KUKA KRL program: MyProgram_054().src

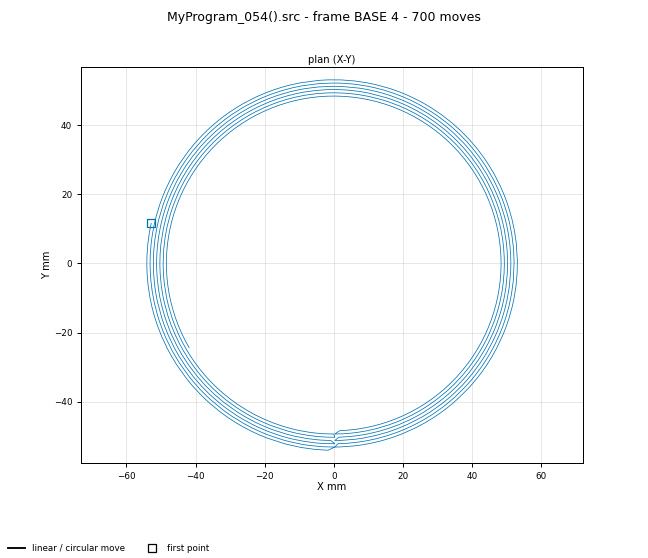
[picture p0: tool path of MyProgram_054().src in frame BASE 4, 700 of 700 moves have a stored position in this frame; points joined in program order, loops and branches not executed]
&ACCESS RVP
&REL 1
&PARAM TEMPLATE = C:\KRC\Roboter\Template\vorgabe
&PARAM EDITMASK = *
DEF MyProgram_054()
; ---- Setting reference (Base) ----
$BASE = BASE_DATA[4]

; --------------------------
; ---- Setting tool (TCP) ----
$TOOL = TOOL_DATA[3]
; --------------------------

$VEL.CP = VEL_APROX_PRINT
Startdeposition()
$VEL.CP = VEL_PRINT
LIN {X -52.8354,Y 11.6366,Z 68,A 162.012,B 24.8649,C -2.6823,E1 24.8431,E2 281.6804} C_DIS
LIN {X -53.3099,Y 9.2261,Z 68,A 164.3906,B 24.8661,C -2.6707,E1 24.8419,E2 279.3155} C_DIS
LIN {X -53.7896,Y 5.8042,Z 68,A 168.8053,B 24.8661,C -2.6709,E1 24.8404,E2 274.8737} C_DIS
LIN {X -54.0573,Y 2.193,Z 68,A 172.1652,B 24.868,C -2.6514,E1 24.8398,E2 271.5403} C_DIS
LIN {X -54.0947,Y -0.8691,Z 68,A 175.1398,B 24.8694,C -2.637,E1 24.8398,E2 268.5822} C_DIS
LIN {X -54.0113,Y -3.1274,Z 68,A 178.3127,B 24.869,C -2.6417,E1 24.8403,E2 265.379} C_DIS
LIN {X -53.6944,Y -6.6329,Z 68,A -178.5265,B 24.871,C -2.6212,E1 24.8412,E2 262.2483} C_DIS
LIN {X -53.1738,Y -9.9794,Z 68,A -174.808,B 24.8719,C -2.6123,E1 24.843,E2 258.5291} C_DIS
LIN {X -52.5931,Y -12.6871,Z 68,A -171.9255,B 24.8728,C -2.6027,E1 24.8447,E2 255.6527} C_DIS
LIN {X -51.9194,Y -15.2111,Z 68,A -168.9774,B 24.8733,C -2.5973,E1 24.847,E2 252.7003} C_DIS
LIN {X -51.0705,Y -17.8546,Z 68,A -165.794,B 24.8738,C -2.5926,E1 24.8498,E2 249.5099} C_DIS
LIN {X -49.8173,Y -21.1005,Z 68,A -162.2259,B 24.875,C -2.5803,E1 24.8536,E2 245.9513} C_DIS
LIN {X -48.2197,Y -24.5327,Z 68,A -158.7451,B 24.8769,C -2.5608,E1 24.8578,E2 242.4982} C_DIS
LIN {X -46.9289,Y -26.9196,Z 68,A -155.3829,B 24.8769,C -2.5611,E1 24.8623,E2 239.1177} C_DIS
LIN {X -45.5694,Y -29.1619,Z 68,A -152.0342,B 24.8766,C -2.5634,E1 24.8674,E2 235.7465} C_DIS
LIN {X -42.5728,Y -33.3851,Z 68,A -147.3331,B 24.8792,C -2.5373,E1 24.8751,E2 231.0852} C_DIS
LIN {X -40.8731,Y -35.4458,Z 68,A -143.9437,B 24.8789,C -2.5402,E1 24.8813,E2 227.6733} C_DIS
LIN {X -38.1407,Y -38.3706,Z 68,A -139.9381,B 24.8801,C -2.5273,E1 24.889,E2 223.6812} C_DIS
LIN {X -35.9398,Y -40.4394,Z 68,A -136.458,B 24.8802,C -2.5259,E1 24.8962,E2 220.1906} C_DIS
LIN {X -32.7163,Y -43.0888,Z 68,A -132.5105,B 24.8818,C -2.5099,E1 24.9048,E2 216.2666} C_DIS
LIN {X -30.733,Y -44.5252,Z 68,A -129.8491,B 24.882,C -2.5068,E1 24.9109,E2 213.6032} C_DIS
LIN {X -28.679,Y -45.8748,Z 68,A -127.1472,B 24.8822,C -2.5046,E1 24.9173,E2 210.8979} C_DIS
LIN {X -26.1922,Y -47.3392,Z 68,A -124.1747,B 24.8828,C -2.499,E1 24.9245,E2 207.9302} C_DIS
LIN {X -23.9334,Y -48.5199,Z 68,A -121.4558,B 24.8831,C -2.496,E1 24.9312,E2 205.2109} C_DIS
LIN {X -21.574,Y -49.614,Z 68,A -118.737,B 24.8834,C -2.4924,E1 24.9382,E2 202.4942} C_DIS
LIN {X -19.3311,Y -50.5304,Z 68,A -115.5128,B 24.8825,C -2.5019,E1 24.9466,E2 199.2404} C_DIS
LIN {X -14.037,Y -52.2489,Z 68,A -109.7546,B 24.8831,C -2.4953,E1 24.962,E2 193.4882} C_DIS
LIN {X -9.435,Y -53.2727,Z 68,A -104.9042,B 24.8836,C -2.4907,E1 24.9753,E2 188.6434} C_DIS
LIN {X -5.5823,Y -53.8128,Z 68,A -101.1152,B 24.8842,C -2.4837,E1 24.9857,E2 184.8682} C_DIS
LIN {X -1.6499,Y -54.0764,Z 68,A -96.3665,B 24.8832,C -2.495,E1 24.999,E2 180.0914} C_DIS
LIN {X -1.6499,Y -54.0764,Z 68,A -96.3665,B 24.8832,C -2.495,E1 24.999,E2 180.0914} C_DIS
Enddeposition()
LIN {X 0.3278,Y -53.1475,Z 68,A -95.9373,B 24.8845,C -2.4803,E1 25.0002,E2 179.6973} C_DIS
Startdeposition()
$VEL.CP = VEL_PRINT
LIN {X -3.2141,Y -53.0599,Z 68,A -100.1608,B 24.8853,C -2.4723,E1 24.9883,E2 183.9405} C_DIS
LIN {X -7.0942,Y -52.683,Z 68,A -104.7462,B 24.8859,C -2.466,E1 24.9755,E2 188.544} C_DIS
LIN {X -9.5086,Y -52.3006,Z 68,A -108.0099,B 24.8868,C -2.4559,E1 24.9665,E2 191.8352} C_DIS
LIN {X -12.9502,Y -51.5571,Z 68,A -110.4894,B 24.8845,C -2.4808,E1 24.9599,E2 194.2587} C_DIS
LIN {X -14.8809,Y -51.0331,Z 68,A -113.3593,B 24.8855,C -2.4697,E1 24.9521,E2 197.1596} C_DIS
LIN {X -19.1384,Y -49.5941,Z 68,A -117.5354,B 24.8841,C -2.4853,E1 24.9412,E2 201.3068} C_DIS
LIN {X -20.8488,Y -48.8986,Z 68,A -119.7452,B 24.8842,C -2.4836,E1 24.9355,E2 203.5258} C_DIS
LIN {X -23.6235,Y -47.6202,Z 68,A -122.6985,B 24.8833,C -2.4931,E1 24.9281,E2 206.4639} C_DIS
LIN {X -25.8654,Y -46.4407,Z 68,A -126.1282,B 24.8841,C -2.4849,E1 24.9196,E2 209.9228} C_DIS
LIN {X -29.6498,Y -44.1209,Z 68,A -130.8923,B 24.8834,C -2.4925,E1 24.9084,E2 214.6841} C_DIS
LIN {X -32.0346,Y -42.4208,Z 68,A -133.8914,B 24.8826,C -2.5004,E1 24.9017,E2 217.675} C_DIS
LIN {X -35.7073,Y -39.3801,Z 68,A -138.5876,B 24.8811,C -2.5172,E1 24.8917,E2 222.3493} C_DIS
LIN {X -36.9563,Y -38.2099,Z 68,A -141.2152,B 24.8819,C -2.5084,E1 24.8864,E2 225.0088} C_DIS
LIN {X -38.8214,Y -36.3135,Z 68,A -144.3826,B 24.8818,C -2.5098,E1 24.8803,E2 228.1866} C_DIS
LIN {X -41.5438,Y -33.1652,Z 68,A -149.0216,B 24.881,C -2.5177,E1 24.8721,E2 232.8282} C_DIS
LIN {X -44.6409,Y -28.8612,Z 68,A -153.9255,B 24.8785,C -2.5444,E1 24.8644,E2 237.6928} C_DIS
LIN {X -46.6361,Y -25.5121,Z 68,A -158.0676,B 24.8773,C -2.5563,E1 24.8586,E2 241.828} C_DIS
LIN {X -48.5908,Y -21.5562,Z 68,A -162.5442,B 24.8757,C -2.5736,E1 24.8532,E2 246.2874} C_DIS
LIN {X -49.5481,Y -19.255,Z 68,A -166.0559,B 24.8761,C -2.5687,E1 24.8495,E2 249.8304} C_DIS
LIN {X -50.5169,Y -16.548,Z 68,A -168.542,B 24.8744,C -2.5869,E1 24.8473,E2 252.2871} C_DIS
LIN {X -51.0383,Y -14.86,Z 68,A -170.8942,B 24.8744,C -2.5859,E1 24.8455,E2 254.6555} C_DIS
LIN {X -51.9733,Y -11.1608,Z 68,A -174.9502,B 24.8732,C -2.5991,E1 24.8429,E2 258.7036} C_DIS
LIN {X -52.5477,Y -8.0316,Z 68,A -178.1632,B 24.8718,C -2.6128,E1 24.8414,E2 261.9029} C_DIS
LIN {X -52.8915,Y -5.3189,Z 68,A 178.4615,B 24.8715,C -2.6156,E1 24.8403,E2 265.2917} C_DIS
LIN {X -53.1233,Y -1.9391,Z 68,A 175.4732,B 24.8694,C -2.6369,E1 24.8399,E2 268.2472} C_DIS
LIN {X -53.1601,Y 0.0529,Z 68,A 172.873,B 24.8694,C -2.6369,E1 24.8398,E2 270.863} C_DIS
LIN {X -53.0965,Y 2.556,Z 68,A 170.427,B 24.8682,C -2.6492,E1 24.84,E2 273.2944} C_DIS
LIN {X -52.8666,Y 5.5568,Z 68,A 166.6141,B 24.868,C -2.651,E1 24.841,E2 277.1258} C_DIS
LIN {X -52.4792,Y 8.4698,Z 68,A 163.9542,B 24.8663,C -2.6684,E1 24.8421,E2 279.7599} C_DIS
LIN {X -51.927,Y 11.3728,Z 68,A 160.5162,B 24.8657,C -2.6746,E1 24.844,E2 283.2033} C_DIS
LIN {X -51.4139,Y 13.5062,Z 68,A 157.8997,B 24.8653,C -2.6782,E1 24.8458,E2 285.8264} C_DIS
LIN {X -50.3836,Y 16.9485,Z 68,A 154.4414,B 24.8635,C -2.6962,E1 24.8487,E2 289.2616} C_DIS
LIN {X -49.6051,Y 19.1074,Z 68,A 151.9867,B 24.8627,C -2.704,E1 24.8511,E2 291.7116} C_DIS
LIN {X -48.8607,Y 20.9401,Z 68,A 149.1689,B 24.8631,C -2.7001,E1 24.8542,E2 294.5542} C_DIS
LIN {X -47.322,Y 24.2153,Z 68,A 146.0235,B 24.8608,C -2.7228,E1 24.858,E2 297.6625} C_DIS
LIN {X -45.9831,Y 26.6713,Z 68,A 142.3868,B 24.8608,C -2.722,E1 24.863,E2 301.3201} C_DIS
LIN {X -44.6959,Y 28.7757,Z 68,A 139.5821,B 24.8603,C -2.7271,E1 24.8672,E2 304.1267} C_DIS
LIN {X -41.9602,Y 32.6366,Z 68,A 134.9399,B 24.8582,C -2.7476,E1 24.8748,E2 308.7425} C_DIS
LIN {X -40.086,Y 34.9123,Z 68,A 131.5433,B 24.8577,C -2.7523,E1 24.8809,E2 312.1434} C_DIS
LIN {X -38.318,Y 36.8441,Z 68,A 129.0783,B 24.8564,C -2.7647,E1 24.8856,E2 314.5896} C_DIS
LIN {X -36.5459,Y 38.6028,Z 68,A 125.9836,B 24.8564,C -2.7647,E1 24.8918,E2 317.6972} C_DIS
LIN {X -34.6267,Y 40.3334,Z 68,A 123.5804,B 24.8552,C -2.7768,E1 24.8968,E2 320.0809} C_DIS
LIN {X -32.3135,Y 42.2093,Z 68,A 119.7034,B 24.8556,C -2.7731,E1 24.9054,E2 323.9811} C_DIS
LIN {X -30.2083,Y 43.7406,Z 68,A 117.2036,B 24.8545,C -2.7835,E1 24.9111,E2 326.4648} C_DIS
LIN {X -27.7183,Y 45.359,Z 68,A 113.9364,B 24.854,C -2.7883,E1 24.9188,E2 329.7308} C_DIS
LIN {X -25.7317,Y 46.5153,Z 68,A 111.2936,B 24.8538,C -2.7899,E1 24.9252,E2 332.3775} C_DIS
LIN {X -22.4129,Y 48.2018,Z 68,A 107.5897,B 24.8526,C -2.8011,E1 24.9345,E2 336.0642} C_DIS
LIN {X -19.7532,Y 49.3519,Z 68,A 104.3841,B 24.8523,C -2.8041,E1 24.9427,E2 339.27} C_DIS
LIN {X -17.1626,Y 50.3114,Z 68,A 101.401,B 24.8519,C -2.8077,E1 24.9506,E2 342.2505} C_DIS
LIN {X -15.0241,Y 50.9906,Z 68,A 99.3463,B 24.851,C -2.8165,E1 24.956,E2 344.2877} C_DIS
LIN {X -12.6183,Y 51.6385,Z 68,A 95.8727,B 24.8521,C -2.8058,E1 24.9655,E2 347.7918} C_DIS
LIN {X -9.8143,Y 52.2445,Z 68,A 92.5219,B 24.8523,C -2.8038,E1 24.9747,E2 351.151} C_DIS
LIN {X -4.2202,Y 52.99,Z 68,A 87.5611,B 24.8499,C -2.8266,E1 24.9883,E2 356.0607} C_DIS
LIN {X -1.6751,Y 53.1314,Z 68,A 83.82,B 24.8517,C -2.8101,E1 24.9989,E2 359.842} C_DIS
LIN {X 2.1559,Y 53.1142,Z 68,A 79.9238,B 24.8512,C -2.8147,E1 25.0097,E2 363.7266} C_DIS
LIN {X 5.9064,Y 52.8292,Z 68,A 76.491,B 24.85,C -2.8255,E1 25.0192,E2 367.1316} C_DIS
LIN {X 9.6926,Y 52.2675,Z 68,A 72.1877,B 24.8505,C -2.821,E1 25.0311,E2 371.4414} C_DIS
LIN {X 12.1047,Y 51.761,Z 68,A 69.0488,B 24.8516,C -2.8108,E1 25.0397,E2 374.6003} C_DIS
LIN {X 16.149,Y 50.646,Z 68,A 65.1105,B 24.8508,C -2.8186,E1 25.0502,E2 378.5135} C_DIS
LIN {X 17.9779,Y 50.0259,Z 68,A 63.0828,B 24.8508,C -2.8178,E1 25.0555,E2 380.5389} C_DIS
LIN {X 19.5219,Y 49.4435,Z 68,A 61.1744,B 24.8513,C -2.8137,E1 25.0605,E2 382.453} C_DIS
LIN {X 21.6172,Y 48.5645,Z 68,A 58.573,B 24.8519,C -2.8081,E1 25.0672,E2 385.0613} C_DIS
LIN {X 24.481,Y 47.1862,Z 68,A 55.3895,B 24.8519,C -2.8086,E1 25.0751,E2 388.2352} C_DIS
LIN {X 26.0526,Y 46.336,Z 68,A 53.2142,B 24.8526,C -2.8012,E1 25.0804,E2 390.4217} C_DIS
LIN {X 28.5062,Y 44.8688,Z 68,A 49.6566,B 24.8541,C -2.7873,E1 25.0889,E2 394.0008} C_DIS
LIN {X 31.3268,Y 42.9464,Z 68,A 46.1605,B 24.8543,C -2.7848,E1 25.0969,E2 397.4907} C_DIS
LIN {X 34.159,Y 40.7305,Z 68,A 42.347,B 24.8549,C -2.7789,E1 25.1051,E2 401.3037} C_DIS
LIN {X 36.7493,Y 38.4094,Z 68,A 38.7438,B 24.8554,C -2.7743,E1 25.1125,E2 404.903} C_DIS
LIN {X 39.3465,Y 35.7446,Z 68,A 34.8229,B 24.8561,C -2.7675,E1 25.12,E2 408.823} C_DIS
LIN {X 41.48,Y 33.2452,Z 68,A 31.8259,B 24.8558,C -2.7705,E1 25.1253,E2 411.7992} C_DIS
LIN {X 43.47,Y 30.5968,Z 68,A 28.2741,B 24.8567,C -2.7623,E1 25.1313,E2 415.3534} C_DIS
LIN {X 44.8639,Y 28.5132,Z 68,A 24.8197,B 24.859,C -2.74,E1 25.1366,E2 418.8433} C_DIS
LIN {X 46.3607,Y 26.0086,Z 68,A 21.4071,B 24.8604,C -2.7262,E1 25.1413,E2 422.2708} C_DIS
LIN {X 48.1892,Y 22.44,Z 68,A 18.0737,B 24.8595,C -2.7349,E1 25.1454,E2 425.5658} C_DIS
LIN {X 49.1769,Y 20.184,Z 68,A 15.2814,B 24.8606,C -2.7246,E1 25.1484,E2 428.3673} C_DIS
LIN {X 50.0014,Y 18.0457,Z 68,A 12.9638,B 24.861,C -2.7207,E1 25.1507,E2 430.6812} C_DIS
LIN {X 50.5399,Y 16.4769,Z 68,A 10.7763,B 24.8624,C -2.707,E1 25.1527,E2 432.8887} C_DIS
LIN {X 51.5927,Y 12.8059,Z 68,A 6.4948,B 24.864,C -2.6913,E1 25.1558,E2 437.1829} C_DIS
LIN {X 52.3205,Y 9.3978,Z 68,A 3.1863,B 24.8642,C -2.6893,E1 25.1576,E2 440.4767} C_DIS
LIN {X 52.8258,Y 5.9371,Z 68,A -1.0908,B 24.8664,C -2.6669,E1 25.1591,E2 444.7816} C_DIS
LIN {X 53.1526,Y 0.7627,Z 68,A -6.8833,B 24.8686,C -2.645,E1 25.1598,E2 450.5912} C_DIS
LIN {X 53.0807,Y -2.8638,Z 68,A -10.392,B 24.869,C -2.6412,E1 25.1594,E2 454.0882} C_DIS
LIN {X 52.7464,Y -6.6049,Z 68,A -14.3544,B 24.8701,C -2.6302,E1 25.1582,E2 458.053} C_DIS
LIN {X 52.1822,Y -10.1383,Z 68,A -18.1421,B 24.8712,C -2.6196,E1 25.1564,E2 461.8437} C_DIS
LIN {X 51.6671,Y -12.501,Z 68,A -20.6513,B 24.8718,C -2.6135,E1 25.1548,E2 464.3526} C_DIS
LIN {X 50.6763,Y -16.0552,Z 68,A -24.1203,B 24.8718,C -2.6121,E1 25.1521,E2 467.8053} C_DIS
LIN {X 49.8631,Y -18.425,Z 68,A -27.481,B 24.8741,C -2.5898,E1 25.1489,E2 471.1997} C_DIS
LIN {X 48.9887,Y -20.6365,Z 68,A -30.1665,B 24.8751,C -2.5796,E1 25.146,E2 473.8947} C_DIS
LIN {X 47.185,Y -24.4833,Z 68,A -34.2041,B 24.8753,C -2.5776,E1 25.1411,E2 477.9154} C_DIS
LIN {X 45.7243,Y -27.1118,Z 68,A -37.4937,B 24.8763,C -2.5674,E1 25.1365,E2 481.2121} C_DIS
LIN {X 44.4237,Y -29.1942,Z 68,A -39.8907,B 24.8765,C -2.5653,E1 25.1329,E2 483.6021} C_DIS
LIN {X 43.1358,Y -31.0663,Z 68,A -42.5014,B 24.8774,C -2.5552,E1 25.1287,E2 486.2237} C_DIS
LIN {X 41.6082,Y -33.0838,Z 68,A -45.2315,B 24.8781,C -2.548,E1 25.124,E2 488.958} C_DIS
LIN {X 40.1285,Y -34.8637,Z 68,A -47.5905,B 24.8785,C -2.5445,E1 25.1197,E2 491.3145} C_DIS
LIN {X 38.842,Y -36.2916,Z 68,A -50.2069,B 24.88,C -2.5281,E1 25.1147,E2 493.9582} C_DIS
LIN {X 35.796,Y -39.2991,Z 68,A -54.0432,B 24.8795,C -2.5333,E1 25.1071,E2 497.7664} C_DIS
LIN {X 34.3492,Y -40.5699,Z 68,A -56.2806,B 24.8803,C -2.5254,E1 25.1023,E2 500.0139} C_DIS
LIN {X 32.5435,Y -42.032,Z 68,A -58.9056,B 24.881,C -2.5175,E1 25.0966,E2 502.6475} C_DIS
LIN {X 30.4989,Y -43.5386,Z 68,A -61.6361,B 24.8815,C -2.5121,E1 25.0904,E2 505.3813} C_DIS
LIN {X 28.602,Y -44.8073,Z 68,A -63.9746,B 24.8818,C -2.5099,E1 25.0849,E2 507.7174} C_DIS
LIN {X 26.4883,Y -46.0882,Z 68,A -67.0071,B 24.8829,C -2.4977,E1 25.0775,E2 510.7694} C_DIS
LIN {X 23.8228,Y -47.5214,Z 68,A -70.3647,B 24.8836,C -2.4905,E1 25.0692,E2 514.1349} C_DIS
LIN {X 19.8322,Y -49.3203,Z 68,A -74.2061,B 24.8826,C -2.5008,E1 25.0595,E2 517.9425} C_DIS
LIN {X 16.7124,Y -50.4632,Z 68,A -78.1833,B 24.8838,C -2.4885,E1 25.049,E2 521.9409} C_DIS
LIN {X 14.0975,Y -51.2547,Z 68,A -81.1698,B 24.8841,C -2.4844,E1 25.0409,E2 524.9319} C_DIS
LIN {X 11.5851,Y -51.8807,Z 68,A -83.8242,B 24.8841,C -2.4844,E1 25.0337,E2 527.5826} C_DIS
LIN {X 8.2617,Y -52.5118,Z 68,A -87.6538,B 24.8847,C -2.478,E1 25.0232,E2 531.423} C_DIS
LIN {X 5.8899,Y -52.8303,Z 68,A -90.5802,B 24.8855,C -2.47,E1 25.015,E2 534.3663} C_DIS
LIN {X 1.7317,Y -53.1297,Z 68,A -94.4063,B 24.8845,C -2.4805,E1 25.0044,E2 538.1659} C_DIS
LIN {X 0.3278,Y -53.1475,Z 68,A -95.9366,B 24.8845,C -2.48,E1 25.0002,E2 539.6973} C_DIS
Enddeposition()
LIN {X 0.3278,Y -53.1475,Z 68,A -95.9366,B 24.8845,C -2.48,E1 25.0002,E2 539.6973} C_DIS
Startdeposition()
$VEL.CP = VEL_PRINT
LIN {X 1.2007,Y -52.2008,Z 68,A -93.7724,B 24.8809,C -2.5188,E1 25.0065,E2 537.4412} C_DIS
LIN {X 3.7036,Y -52.0819,Z 68,A -91.0856,B 24.8809,C -2.5188,E1 25.0139,E2 534.7556} C_DIS
LIN {X 6.9902,Y -51.7448,Z 68,A -87.899,B 24.8815,C -2.5126,E1 25.0227,E2 531.5859} C_DIS
LIN {X 9.5939,Y -51.3254,Z 68,A -84.4131,B 24.8802,C -2.5261,E1 25.0324,E2 528.0716} C_DIS
LIN {X 12.2252,Y -50.763,Z 68,A -81.8964,B 24.8808,C -2.5204,E1 25.0392,E2 525.5718} C_DIS
LIN {X 15.4906,Y -49.8633,Z 68,A -78.0208,B 24.8801,C -2.5276,E1 25.0496,E2 521.6859} C_DIS
LIN {X 18.3377,Y -48.8883,Z 68,A -74.7631,B 24.8798,C -2.5309,E1 25.0582,E2 518.4269} C_DIS
LIN {X 20.4504,Y -48.0429,Z 68,A -72.3518,B 24.8796,C -2.5327,E1 25.0644,E2 516.0168} C_DIS
LIN {X 22.4531,Y -47.1401,Z 68,A -69.8259,B 24.879,C -2.5387,E1 25.0708,E2 513.4832} C_DIS
LIN {X 24.1625,Y -46.2874,Z 68,A -67.9284,B 24.879,C -2.5382,E1 25.0755,E2 511.5921} C_DIS
LIN {X 26.2875,Y -45.1148,Z 68,A -65.0106,B 24.8781,C -2.548,E1 25.0826,E2 508.6599} C_DIS
LIN {X 28.7287,Y -43.6001,Z 68,A -61.8105,B 24.8775,C -2.5549,E1 25.0902,E2 505.4537} C_DIS
LIN {X 31.3281,Y -41.7715,Z 68,A -58.6989,B 24.8775,C -2.5543,E1 25.0972,E2 502.3545} C_DIS
LIN {X 32.8885,Y -40.5544,Z 68,A -55.8361,B 24.8757,C -2.5732,E1 25.1035,E2 499.4578} C_DIS
LIN {X 35.0118,Y -38.7368,Z 68,A -52.7354,B 24.875,C -2.5808,E1 25.11,E2 496.3514} C_DIS
LIN {X 38.2717,Y -35.5199,Z 68,A -48.6469,B 24.8757,C -2.5734,E1 25.1179,E2 492.2979} C_DIS
LIN {X 40.1139,Y -33.4244,Z 68,A -45.4119,B 24.8746,C -2.5848,E1 25.1238,E2 489.0506} C_DIS
LIN {X 41.3473,Y -31.8858,Z 68,A -42.9646,B 24.8734,C -2.5964,E1 25.1281,E2 486.5874} C_DIS
LIN {X 43.203,Y -29.3225,Z 68,A -39.5516,B 24.8726,C -2.6045,E1 25.1336,E2 483.1718} C_DIS
LIN {X 44.7418,Y -26.9172,Z 68,A -36.3924,B 24.8717,C -2.6138,E1 25.1382,E2 480.0067} C_DIS
LIN {X 45.9347,Y -24.8258,Z 68,A -34.2432,B 24.872,C -2.611,E1 25.1411,E2 477.8754} C_DIS
LIN {X 46.8178,Y -23.1172,Z 68,A -31.8383,B 24.8708,C -2.6233,E1 25.1442,E2 475.454} C_DIS
LIN {X 48.0762,Y -20.3714,Z 68,A -28.7816,B 24.8704,C -2.6277,E1 25.1476,E2 472.4037} C_DIS
LIN {X 48.9685,Y -18.1232,Z 68,A -25.588,B 24.8684,C -2.6472,E1 25.1508,E2 469.1817} C_DIS
LIN {X 49.8838,Y -15.4247,Z 68,A -22.5315,B 24.8676,C -2.6553,E1 25.1534,E2 466.1234} C_DIS
LIN {X 50.6755,Y -12.5838,Z 68,A -19.3049,B 24.8666,C -2.6651,E1 25.1557,E2 462.8921} C_DIS
LIN {X 51.4366,Y -8.9803,Z 68,A -15.5277,B 24.8659,C -2.6721,E1 25.1577,E2 459.1205} C_DIS
LIN {X 51.9731,Y -5.0149,Z 68,A -10.3276,B 24.8628,C -2.7034,E1 25.1594,E2 453.8772} C_DIS
LIN {X 52.2139,Y 0.3513,Z 68,A -4.5685,B 24.8612,C -2.719,E1 25.1597,E2 448.1154} C_DIS
LIN {X 52.0275,Y 4.4168,Z 68,A -0.3147,B 24.8602,C -2.7283,E1 25.1589,E2 443.8647} C_DIS
LIN {X 51.5536,Y 8.2844,Z 68,A 3.549,B 24.8597,C -2.7327,E1 25.1573,E2 440.0135} C_DIS
LIN {X 50.8864,Y 11.6998,Z 68,A 7.0648,B 24.8592,C -2.7379,E1 25.1553,E2 436.5059} C_DIS
LIN {X 50.2849,Y 14.0622,Z 68,A 10.0343,B 24.8577,C -2.7521,E1 25.1532,E2 433.5198} C_DIS
LIN {X 49.4397,Y 16.7941,Z 68,A 12.8575,B 24.8575,C -2.7546,E1 25.1507,E2 430.7066} C_DIS
LIN {X 48.7669,Y 18.6582,Z 68,A 14.8622,B 24.8572,C -2.7573,E1 25.1488,E2 428.7068} C_DIS
LIN {X 47.7195,Y 21.1952,Z 68,A 18.4495,B 24.8551,C -2.7779,E1 25.1448,E2 425.0905} C_DIS
LIN {X 46.144,Y 24.4343,Z 68,A 22.4166,B 24.8539,C -2.7889,E1 25.1398,E2 421.1184} C_DIS
LIN {X 44.0565,Y 28.0234,Z 68,A 26.713,B 24.8532,C -2.7952,E1 25.1336,E2 416.8288} C_DIS
LIN {X 42.4536,Y 30.3974,Z 68,A 30.2406,B 24.8516,C -2.8109,E1 25.1279,E2 413.2813} C_DIS
LIN {X 40.5493,Y 32.8947,Z 68,A 33.4134,B 24.8513,C -2.8133,E1 25.1224,E2 410.1177} C_DIS
LIN {X 38.6742,Y 35.0814,Z 68,A 36.2791,B 24.8513,C -2.8143,E1 25.1171,E2 407.2625} C_DIS
LIN {X 36.2281,Y 37.601,Z 68,A 39.8075,B 24.8511,C -2.8158,E1 25.1102,E2 403.7455} C_DIS
LIN {X 34.4102,Y 39.2715,Z 68,A 42.7374,B 24.85,C -2.8255,E1 25.1041,E2 400.8043} C_DIS
LIN {X 32.7671,Y 40.6527,Z 68,A 45.8391,B 24.848,C -2.8448,E1 25.0973,E2 397.6687} C_DIS
LIN {X 29.8757,Y 42.8224,Z 68,A 49.1443,B 24.8487,C -2.8383,E1 25.0898,E2 394.3905} C_DIS
LIN {X 27.988,Y 44.08,Z 68,A 51.7817,B 24.8479,C -2.845,E1 25.0836,E2 391.7458} C_DIS
LIN {X 24.7155,Y 45.9945,Z 68,A 55.7511,B 24.8477,C -2.847,E1 25.074,E2 387.7834} C_DIS
LIN {X 22.1577,Y 47.2796,Z 68,A 58.8989,B 24.8473,C -2.8509,E1 25.0661,E2 384.6346} C_DIS
LIN {X 19.7851,Y 48.3205,Z 68,A 61.7258,B 24.847,C -2.8535,E1 25.0588,E2 381.8082} C_DIS
LIN {X 17.2309,Y 49.289,Z 68,A 64.6932,B 24.8468,C -2.8557,E1 25.051,E2 378.842} C_DIS
LIN {X 14.4825,Y 50.1661,Z 68,A 67.922,B 24.8464,C -2.8591,E1 25.0424,E2 375.6106} C_DIS
LIN {X 11.9937,Y 50.8176,Z 68,A 70.7137,B 24.8464,C -2.8602,E1 25.0348,E2 372.8206} C_DIS
LIN {X 10.021,Y 51.2436,Z 68,A 72.93,B 24.8462,C -2.8611,E1 25.0288,E2 370.6046} C_DIS
LIN {X 6.9548,Y 51.7494,Z 68,A 76.043,B 24.8467,C -2.8567,E1 25.0202,E2 367.5052} C_DIS
LIN {X 5.4409,Y 51.9298,Z 68,A 78.0087,B 24.8461,C -2.8622,E1 25.0147,E2 365.5277} C_DIS
LIN {X 2.4355,Y 52.1576,Z 68,A 81.2381,B 24.8462,C -2.8608,E1 25.0057,E2 362.3029} C_DIS
LIN {X -0.237,Y 52.2136,Z 68,A 84.7379,B 24.8452,C -2.8704,E1 24.9959,E2 358.7805} C_DIS
LIN {X -4.4458,Y 52.0252,Z 68,A 89.4616,B 24.8452,C -2.8703,E1 24.9827,E2 354.0553} C_DIS
LIN {X -9.1801,Y 51.4008,Z 68,A 94.127,B 24.8467,C -2.8568,E1 24.9699,E2 349.4181} C_DIS
LIN {X -11.9273,Y 50.8339,Z 68,A 97.6428,B 24.8461,C -2.8616,E1 24.9603,E2 345.8863} C_DIS
LIN {X -14.9887,Y 50.0164,Z 68,A 100.8953,B 24.847,C -2.8541,E1 24.9516,E2 342.6464} C_DIS
LIN {X -18.2145,Y 48.9347,Z 68,A 104.3166,B 24.848,C -2.8443,E1 24.9427,E2 339.2418} C_DIS
LIN {X -20.4534,Y 48.0417,Z 68,A 106.8717,B 24.8486,C -2.8392,E1 24.9361,E2 336.6932} C_DIS
LIN {X -22.2243,Y 47.2486,Z 68,A 109.6359,B 24.8478,C -2.8464,E1 24.929,E2 333.9047} C_DIS
LIN {X -25.0712,Y 45.8016,Z 68,A 112.3861,B 24.8497,C -2.8284,E1 24.9223,E2 331.19} C_DIS
LIN {X -26.937,Y 44.7298,Z 68,A 116.0793,B 24.8478,C -2.8458,E1 24.9133,E2 327.4439} C_DIS
LIN {X -29.6438,Y 42.9836,Z 68,A 118.1309,B 24.8511,C -2.8152,E1 24.9087,E2 325.4587} C_DIS
LIN {X -31.4396,Y 41.6877,Z 68,A 121.0877,B 24.8508,C -2.8186,E1 24.902,E2 322.4831} C_DIS
LIN {X -33.7792,Y 39.8156,Z 68,A 123.8326,B 24.8524,C -2.803,E1 24.8962,E2 319.7651} C_DIS
LIN {X -35.8205,Y 37.9895,Z 68,A 127.8827,B 24.8514,C -2.8126,E1 24.8877,E2 315.6758} C_DIS
LIN {X -37.868,Y 35.9497,Z 68,A 131.1106,B 24.8521,C -2.8058,E1 24.8815,E2 312.4501} C_DIS
LIN {X -40.9903,Y 32.3435,Z 68,A 135.348,B 24.8551,C -2.7772,E1 24.874,E2 308.2618} C_DIS
LIN {X -42.5301,Y 30.2902,Z 68,A 139.0655,B 24.8545,C -2.7835,E1 24.8678,E2 304.5112} C_DIS
LIN {X -44.1197,Y 27.9252,Z 68,A 142.0352,B 24.8556,C -2.7725,E1 24.8633,E2 301.5529} C_DIS
LIN {X -45.9239,Y 24.8457,Z 68,A 145.4828,B 24.8575,C -2.7543,E1 24.8586,E2 298.1307} C_DIS
LIN {X -46.9052,Y 22.941,Z 68,A 148.4228,B 24.8573,C -2.7563,E1 24.8549,E2 295.17} C_DIS
LIN {X -47.9109,Y 20.7573,Z 68,A 150.8147,B 24.8585,C -2.7448,E1 24.8522,E2 292.7925} C_DIS
LIN {X -48.8857,Y 18.3442,Z 68,A 153.3925,B 24.8598,C -2.7321,E1 24.8496,E2 290.2306} C_DIS
LIN {X -49.4483,Y 16.7684,Z 68,A 155.9091,B 24.8593,C -2.7367,E1 24.8473,E2 287.6888} C_DIS
LIN {X -50.6514,Y 12.6825,Z 68,A 160.5516,B 24.8609,C -2.7218,E1 24.8439,E2 283.0549} C_DIS
LIN {X -51.3189,Y 9.6282,Z 68,A 163.7038,B 24.8624,C -2.7069,E1 24.8422,E2 279.9197} C_DIS
LIN {X -51.7597,Y 6.872,Z 68,A 166.8961,B 24.8632,C -2.6992,E1 24.8409,E2 276.7267} C_DIS
LIN {X -52.0814,Y 3.7254,Z 68,A 170.2384,B 24.8645,C -2.6864,E1 24.8401,E2 273.3951} C_DIS
LIN {X -52.2046,Y 0.9956,Z 68,A 173.6641,B 24.8648,C -2.6833,E1 24.8398,E2 269.9562} C_DIS
LIN {X -52.1647,Y -2.2699,Z 68,A 176.8993,B 24.8664,C -2.6668,E1 24.84,E2 266.7408} C_DIS
LIN {X -51.8799,Y -5.9007,Z 68,A -178.518,B 24.8668,C -2.6632,E1 24.8413,E2 262.1393} C_DIS
LIN {X -51.4684,Y -8.7948,Z 68,A -175.7448,B 24.8685,C -2.6468,E1 24.8425,E2 259.3888} C_DIS
LIN {X -51.0492,Y -10.969,Z 68,A -172.8105,B 24.8685,C -2.6471,E1 24.8442,E2 256.4367} C_DIS
LIN {X -49.7332,Y -15.9045,Z 68,A -168.2663,B 24.8717,C -2.6144,E1 24.8476,E2 251.9443} C_DIS
LIN {X -49.045,Y -17.9137,Z 68,A -164.7943,B 24.8706,C -2.625,E1 24.8509,E2 248.4273} C_DIS
LIN {X -47.8972,Y -20.7889,Z 68,A -161.0104,B 24.871,C -2.6214,E1 24.8551,E2 244.6309} C_DIS
LIN {X -46.075,Y -24.5656,Z 68,A -157.3797,B 24.8737,C -2.5939,E1 24.8597,E2 241.0467} C_DIS
LIN {X -44.7087,Y -26.9716,Z 68,A -154.0153,B 24.874,C -2.5911,E1 24.8644,E2 237.6714} C_DIS
LIN {X -42.7042,Y -30.0458,Z 68,A -149.0279,B 24.8734,C -2.5964,E1 24.8724,E2 232.6467} C_DIS
LIN {X -40.5227,Y -32.9275,Z 68,A -145.9912,B 24.8758,C -2.5723,E1 24.8776,E2 229.6534} C_DIS
LIN {X -38.1501,Y -35.6498,Z 68,A -142.8037,B 24.8778,C -2.5512,E1 24.8835,E2 226.5019} C_DIS
LIN {X -35.759,Y -38.0474,Z 68,A -139.1122,B 24.8786,C -2.5432,E1 24.8908,E2 222.814} C_DIS
LIN {X -32.9352,Y -40.5165,Z 68,A -134.8843,B 24.8792,C -2.5371,E1 24.8997,E2 218.584} C_DIS
LIN {X -30.8948,Y -42.093,Z 68,A -131.4388,B 24.8787,C -2.5424,E1 24.9074,E2 215.1136} C_DIS
LIN {X -27.9737,Y -44.0892,Z 68,A -128.0415,B 24.88,C -2.5282,E1 24.9153,E2 211.7388} C_DIS
LIN {X -26.3271,Y -45.0918,Z 68,A -125.4385,B 24.8795,C -2.5334,E1 24.9216,E2 209.1155} C_DIS
LIN {X -23.6104,Y -46.5713,Z 68,A -122.6543,B 24.8809,C -2.5188,E1 24.9284,E2 206.3585} C_DIS
LIN {X -21.6547,Y -47.5124,Z 68,A -119.5684,B 24.88,C -2.5281,E1 24.9362,E2 203.2426} C_DIS
LIN {X -18.9453,Y -48.656,Z 68,A -116.3556,B 24.8803,C -2.5247,E1 24.9446,E2 200.0307} C_DIS
LIN {X -15.9666,Y -49.7127,Z 68,A -113.1831,B 24.8811,C -2.5168,E1 24.9529,E2 196.8711} C_DIS
LIN {X -13.608,Y -50.4096,Z 68,A -110.7445,B 24.8817,C -2.5105,E1 24.9594,E2 194.4436} C_DIS
LIN {X -11.8411,Y -50.8538,Z 68,A -107.9542,B 24.8805,C -2.5235,E1 24.9671,E2 191.6185} C_DIS
LIN {X -8.6106,Y -51.4992,Z 68,A -104.6005,B 24.881,C -2.5176,E1 24.9763,E2 188.2754} C_DIS
LIN {X -5.2253,Y -51.9524,Z 68,A -101.3512,B 24.8819,C -2.5079,E1 24.9852,E2 185.0468} C_DIS
LIN {X -3.3589,Y -52.1062,Z 68,A -98.5237,B 24.8806,C -2.5221,E1 24.9932,E2 182.1846} C_DIS
LIN {X 0.3319,Y -52.2067,Z 68,A -96.1542,B 24.8834,C -2.492,E1 24.9996,E2 179.8863} C_DIS
Enddeposition()
LIN {X 0.3319,Y -52.2067,Z 68,A -96.1542,B 24.8834,C -2.492,E1 24.9996,E2 179.8863} C_DIS
Startdeposition()
$VEL.CP = VEL_PRINT
LIN {X -0.8087,Y -51.2641,Z 68,A -97.7461,B 24.8824,C -2.5026,E1 24.9952,E2 181.4532} C_DIS
LIN {X -3.7459,Y -51.1341,Z 68,A -100.8536,B 24.8822,C -2.5056,E1 24.9866,E2 184.5545} C_DIS
LIN {X -5.5282,Y -50.9717,Z 68,A -102.9078,B 24.8822,C -2.5048,E1 24.9809,E2 186.6117} C_DIS
LIN {X -8.0735,Y -50.6311,Z 68,A -106.1583,B 24.8828,C -2.499,E1 24.9719,E2 189.8789} C_DIS
LIN {X -11.4791,Y -49.9688,Z 68,A -109.6591,B 24.882,C -2.5071,E1 24.9623,E2 193.3647} C_DIS
LIN {X -13.4357,Y -49.4786,Z 68,A -112.2716,B 24.8825,C -2.5024,E1 24.9553,E2 195.9923} C_DIS
LIN {X -17.0996,Y -48.3348,Z 68,A -115.8765,B 24.8811,C -2.5171,E1 24.9458,E2 199.5688} C_DIS
LIN {X -18.7522,Y -47.7179,Z 68,A -117.8059,B 24.8808,C -2.5196,E1 24.9407,E2 201.4964} C_DIS
LIN {X -20.8732,Y -46.8294,Z 68,A -120.9009,B 24.8814,C -2.5136,E1 24.9327,E2 204.6128} C_DIS
LIN {X -23.1559,Y -45.7437,Z 68,A -123.7032,B 24.881,C -2.5173,E1 24.9257,E2 207.4135} C_DIS
LIN {X -25.6921,Y -44.3688,Z 68,A -126.8217,B 24.8805,C -2.5234,E1 24.9182,E2 210.5268} C_DIS
LIN {X -28.124,Y -42.8684,Z 68,A -130.8298,B 24.8812,C -2.5154,E1 24.9087,E2 214.5668} C_DIS
LIN {X -31.806,Y -40.2123,Z 68,A -134.6994,B 24.8786,C -2.5428,E1 24.9001,E2 218.3848} C_DIS
LIN {X -34.5688,Y -37.8636,Z 68,A -138.9491,B 24.8782,C -2.5474,E1 24.8911,E2 222.6402} C_DIS
LIN {X -37.0936,Y -35.3946,Z 68,A -142.748,B 24.8772,C -2.5578,E1 24.8836,E2 226.4303} C_DIS
LIN {X -39.3761,Y -32.8356,Z 68,A -146.9834,B 24.877,C -2.5602,E1 24.8758,E2 230.6791} C_DIS
LIN {X -42.0224,Y -29.3732,Z 68,A -151.8997,B 24.8759,C -2.5711,E1 24.8676,E2 235.5929} C_DIS
LIN {X -43.9944,Y -26.3289,Z 68,A -156.0437,B 24.875,C -2.5801,E1 24.8615,E2 239.7365} C_DIS
LIN {X -45.32,Y -23.9739,Z 68,A -158.8961,B 24.874,C -2.5906,E1 24.8577,E2 242.5789} C_DIS
LIN {X -46.8687,Y -20.7849,Z 68,A -162.6411,B 24.8726,C -2.6047,E1 24.8532,E2 246.3106} C_DIS
LIN {X -47.4227,Y -19.4873,Z 68,A -165.3906,B 24.8738,C -2.5922,E1 24.8502,E2 249.1052} C_DIS
LIN {X -48.7728,Y -15.8068,Z 68,A -168.8073,B 24.8712,C -2.6187,E1 24.8472,E2 252.478} C_DIS
LIN {X -49.6569,Y -12.7608,Z 68,A -172.9324,B 24.871,C -2.621,E1 24.8441,E2 256.6216} C_DIS
LIN {X -50.3229,Y -9.808,Z 68,A -176.1319,B 24.8697,C -2.6339,E1 24.8423,E2 259.8092} C_DIS
LIN {X -50.7273,Y -7.4458,Z 68,A -179.8186,B 24.8703,C -2.628,E1 24.8408,E2 263.5319} C_DIS
LIN {X -51.1133,Y -4.0099,Z 68,A 177.5359,B 24.8674,C -2.657,E1 24.8401,E2 266.1238} C_DIS
LIN {X -51.2514,Y -1.4029,Z 68,A 174.6766,B 24.8664,C -2.667,E1 24.8398,E2 268.9765} C_DIS
LIN {X -51.2622,Y 0.9094,Z 68,A 172.0803,B 24.8656,C -2.675,E1 24.8398,E2 271.5694} C_DIS
LIN {X -51.1841,Y 2.9757,Z 68,A 169.7958,B 24.8649,C -2.6826,E1 24.8401,E2 273.8494} C_DIS
LIN {X -51.0191,Y 5.0758,Z 68,A 167.326,B 24.8643,C -2.6884,E1 24.8407,E2 276.3202} C_DIS
LIN {X -50.644,Y 7.9911,Z 68,A 163.6039,B 24.8639,C -2.6926,E1 24.8422,E2 280.0545} C_DIS
LIN {X -50.1036,Y 10.8755,Z 68,A 160.7027,B 24.8623,C -2.7081,E1 24.8438,E2 282.9356} C_DIS
LIN {X -49.602,Y 12.9745,Z 68,A 158.3301,B 24.8614,C -2.7161,E1 24.8454,E2 285.303} C_DIS
LIN {X -48.9598,Y 15.218,Z 68,A 155.4965,B 24.861,C -2.721,E1 24.8477,E2 288.1413} C_DIS
LIN {X -48.163,Y 17.5775,Z 68,A 152.3392,B 24.8606,C -2.7241,E1 24.8507,E2 291.3089} C_DIS
LIN {X -47.0789,Y 20.3041,Z 68,A 149.1581,B 24.8595,C -2.7352,E1 24.8541,E2 294.4811} C_DIS
LIN {X -45.7787,Y 23.0874,Z 68,A 145.9999,B 24.858,C -2.7491,E1 24.8579,E2 297.6231} C_DIS
LIN {X -44.9116,Y 24.732,Z 68,A 143.8214,B 24.8576,C -2.7536,E1 24.8608,E2 299.8024} C_DIS
LIN {X -43.5554,Y 27.048,Z 68,A 141.1218,B 24.8563,C -2.7663,E1 24.8647,E2 302.4855} C_DIS
LIN {X -42.6401,Y 28.4702,Z 68,A 139.0175,B 24.856,C -2.7684,E1 24.8679,E2 304.5954} C_DIS
LIN {X -40.9737,Y 30.8188,Z 68,A 135.7117,B 24.8553,C -2.7757,E1 24.8733,E2 307.8999} C_DIS
LIN {X -38.5495,Y 33.8022,Z 68,A 131.0811,B 24.8547,C -2.7817,E1 24.8817,E2 312.5374} C_DIS
LIN {X -36.7313,Y 35.7705,Z 68,A 128.1852,B 24.8537,C -2.7904,E1 24.8872,E2 315.4252} C_DIS
LIN {X -33.9447,Y 38.4251,Z 68,A 124.0239,B 24.8525,C -2.8022,E1 24.8957,E2 319.575} C_DIS
LIN {X -31.1612,Y 40.7136,Z 68,A 119.7751,B 24.8519,C -2.8074,E1 24.905,E2 323.8272} C_DIS
LIN {X -29.0309,Y 42.2596,Z 68,A 117.229,B 24.8507,C -2.8192,E1 24.9108,E2 326.3539} C_DIS
LIN {X -27.0508,Y 43.5536,Z 68,A 114.453,B 24.8504,C -2.8221,E1 24.9173,E2 329.1319} C_DIS
LIN {X -24.7912,Y 44.8787,Z 68,A 111.7908,B 24.8494,C -2.8313,E1 24.9237,E2 331.7802} C_DIS
LIN {X -22.5297,Y 46.0557,Z 68,A 108.9982,B 24.8488,C -2.8367,E1 24.9307,E2 334.5673} C_DIS
LIN {X -20.7937,Y 46.8647,Z 68,A 106.5471,B 24.849,C -2.835,E1 24.9369,E2 337.0285} C_DIS
LIN {X -18.8412,Y 47.6829,Z 68,A 104.345,B 24.8484,C -2.8408,E1 24.9426,E2 339.2216} C_DIS
LIN {X -16.2126,Y 48.6398,Z 68,A 100.5211,B 24.8492,C -2.8335,E1 24.9527,E2 343.0704} C_DIS
LIN {X -12.7282,Y 49.6653,Z 68,A 96.9641,B 24.8479,C -2.8458,E1 24.9623,E2 346.6038} C_DIS
LIN {X -10.3193,Y 50.2211,Z 68,A 94.1397,B 24.8477,C -2.8471,E1 24.97,E2 349.4284} C_DIS
LIN {X -8.2819,Y 50.5973,Z 68,A 91.5954,B 24.8479,C -2.845,E1 24.977,E2 351.9802} C_DIS
LIN {X -4.4591,Y 51.0767,Z 68,A 86.5266,B 24.849,C -2.8346,E1 24.9911,E2 357.0765} C_DIS
LIN {X -0.0283,Y 51.271,Z 68,A 82.5726,B 24.8471,C -2.8528,E1 25.0021,E2 360.9877} C_DIS
LIN {X 2.4813,Y 51.211,Z 68,A 79.0899,B 24.8483,C -2.8414,E1 25.0118,E2 364.4966} C_DIS
LIN {X 7.4712,Y 50.7237,Z 68,A 74.156,B 24.8472,C -2.852,E1 25.0254,E2 369.4015} C_DIS
LIN {X 9.9052,Y 50.3048,Z 68,A 71.754,B 24.8466,C -2.8573,E1 25.032,E2 371.7883} C_DIS
LIN {X 12.4115,Y 49.7454,Z 68,A 68.2518,B 24.848,C -2.8446,E1 25.0416,E2 375.3158} C_DIS
LIN {X 14.8769,Y 49.0647,Z 68,A 65.8404,B 24.8473,C -2.8506,E1 25.048,E2 377.7088} C_DIS
LIN {X 16.4811,Y 48.5492,Z 68,A 63.5097,B 24.8484,C -2.841,E1 25.0542,E2 380.0579} C_DIS
LIN {X 20.1701,Y 47.1369,Z 68,A 59.7601,B 24.8475,C -2.8488,E1 25.0639,E2 383.7805} C_DIS
LIN {X 22.4437,Y 46.0977,Z 68,A 56.5745,B 24.8486,C -2.8384,E1 25.072,E2 386.9828} C_DIS
LIN {X 24.744,Y 44.905,Z 68,A 53.3742,B 24.8497,C -2.8289,E1 25.0799,E2 390.1964} C_DIS
LIN {X 27.4699,Y 43.2911,Z 68,A 49.8931,B 24.8501,C -2.8247,E1 25.0882,E2 393.6764} C_DIS
LIN {X 29.9782,Y 41.5934,Z 68,A 46.6007,B 24.8505,C -2.8209,E1 25.0957,E2 396.9665} C_DIS
LIN {X 32.5407,Y 39.6212,Z 68,A 43.4095,B 24.8503,C -2.8225,E1 25.1026,E2 400.142} C_DIS
LIN {X 34.7073,Y 37.7366,Z 68,A 40.0572,B 24.8513,C -2.8135,E1 25.1097,E2 403.5022} C_DIS
LIN {X 37.6447,Y 34.8074,Z 68,A 35.5629,B 24.852,C -2.8066,E1 25.1185,E2 407.9939} C_DIS
LIN {X 39.7733,Y 32.3534,Z 68,A 31.9889,B 24.8528,C -2.7994,E1 25.1249,E2 411.5684} C_DIS
LIN {X 41.434,Y 30.1974,Z 68,A 28.9725,B 24.8535,C -2.7927,E1 25.13,E2 414.5865} C_DIS
LIN {X 42.4862,Y 28.698,Z 68,A 26.2861,B 24.8554,C -2.7749,E1 25.1343,E2 417.3017} C_DIS
LIN {X 44.3654,Y 25.698,Z 68,A 22.2803,B 24.8565,C -2.7637,E1 25.14,E2 421.3137} C_DIS
LIN {X 46.1778,Y 22.277,Z 68,A 18.7732,B 24.856,C -2.7684,E1 25.1445,E2 424.791} C_DIS
LIN {X 47.2402,Y 19.9252,Z 68,A 15.6277,B 24.8574,C -2.755,E1 25.148,E2 427.9509} C_DIS
LIN {X 48.129,Y 17.6706,Z 68,A 12.1343,B 24.8599,C -2.7314,E1 25.1514,E2 431.4807} C_DIS
LIN {X 49.4435,Y 13.5654,Z 68,A 8.127,B 24.8597,C -2.7336,E1 25.1546,E2 435.46} C_DIS
LIN {X 50.0822,Y 10.9737,Z 68,A 5.0214,B 24.8608,C -2.7221,E1 25.1566,E2 438.5748} C_DIS
LIN {X 50.5941,Y 8.3011,Z 68,A 2.1699,B 24.8614,C -2.7166,E1 25.158,E2 441.4225} C_DIS
LIN {X 50.9961,Y 5.2956,Z 68,A -1.2446,B 24.8625,C -2.7056,E1 25.1591,E2 444.8429} C_DIS
LIN {X 51.2094,Y 2.517,Z 68,A -3.9853,B 24.8627,C -2.7035,E1 25.1596,E2 447.5722} C_DIS
LIN {X 51.273,Y -0.0468,Z 68,A -7.5888,B 24.8652,C -2.6793,E1 25.1597,E2 451.2115} C_DIS
LIN {X 51.218,Y -2.3185,Z 68,A -10.2622,B 24.8663,C -2.6686,E1 25.1594,E2 453.8944} C_DIS
LIN {X 50.7461,Y -7.3139,Z 68,A -15.2768,B 24.8668,C -2.6631,E1 25.1578,E2 458.8924} C_DIS
LIN {X 50.078,Y -10.9918,Z 68,A -19.6072,B 24.8684,C -2.6469,E1 25.1555,E2 463.2358} C_DIS
LIN {X 49.4645,Y -13.4877,Z 68,A -22.3393,B 24.869,C -2.6408,E1 25.1536,E2 465.9665} C_DIS
LIN {X 48.6396,Y -16.213,Z 68,A -26.1315,B 24.8713,C -2.6186,E1 25.1503,E2 469.7897} C_DIS
LIN {X 47.4277,Y -19.4751,Z 68,A -28.9406,B 24.8702,C -2.629,E1 25.1475,E2 472.5587} C_DIS
LIN {X 46.3211,Y -21.9762,Z 68,A -32.8582,B 24.8728,C -2.6024,E1 25.1429,E2 476.518} C_DIS
LIN {X 44.1395,Y -26.0835,Z 68,A -37.9181,B 24.874,C -2.5903,E1 25.136,E2 481.5801} C_DIS
LIN {X 42.5304,Y -28.6327,Z 68,A -41.1614,B 24.8747,C -2.5836,E1 25.131,E2 484.8231} C_DIS
LIN {X 40.2989,Y -31.6963,Z 68,A -45.0626,B 24.8751,C -2.5791,E1 25.1244,E2 488.7164} C_DIS
LIN {X 38.4358,Y -33.9318,Z 68,A -48.1128,B 24.8755,C -2.5749,E1 25.1189,E2 491.7627} C_DIS
LIN {X 37.1523,Y -35.3324,Z 68,A -50.5888,B 24.8767,C -2.5626,E1 25.1141,E2 494.2569} C_DIS
LIN {X 34.8216,Y -37.6317,Z 68,A -53.8272,B 24.8767,C -2.5624,E1 25.1076,E2 497.4823} C_DIS
LIN {X 33.4009,Y -38.8978,Z 68,A -56.2661,B 24.8778,C -2.5515,E1 25.1025,E2 499.9376} C_DIS
LIN {X 31.1355,Y -40.734,Z 68,A -59.6725,B 24.8787,C -2.5417,E1 25.095,E2 503.3546} C_DIS
LIN {X 28.0259,Y -42.9331,Z 68,A -63.3691,B 24.8785,C -2.5442,E1 25.0865,E2 507.0326} C_DIS
LIN {X 25.4695,Y -44.4967,Z 68,A -67.5016,B 24.8805,C -2.5231,E1 25.0765,E2 511.2025} C_DIS
LIN {X 21.125,Y -46.716,Z 68,A -72.8313,B 24.8811,C -2.5168,E1 25.0631,E2 516.5329} C_DIS
LIN {X 18.2951,Y -47.8947,Z 68,A -75.881,B 24.8809,C -2.5192,E1 25.0552,E2 519.5703} C_DIS
LIN {X 15.564,Y -48.8514,Z 68,A -79.4253,B 24.8818,C -2.5095,E1 25.0458,E2 523.1308} C_DIS
LIN {X 12.1423,Y -49.8117,Z 68,A -82.8002,B 24.8811,C -2.5164,E1 25.0367,E2 526.4838} C_DIS
LIN {X 8.4057,Y -50.5766,Z 68,A -87.2291,B 24.8818,C -2.5099,E1 25.0246,E2 530.9231} C_DIS
LIN {X 6.048,Y -50.9124,Z 68,A -89.7293,B 24.8816,C -2.5111,E1 25.0176,E2 533.4183} C_DIS
LIN {X 1.8817,Y -51.2367,Z 68,A -94.1965,B 24.8815,C -2.5127,E1 25.0052,E2 537.8798} C_DIS
LIN {X 0.3271,Y -51.2583,Z 68,A -95.6732,B 24.8811,C -2.517,E1 25.0011,E2 539.3459} C_DIS
Enddeposition()
LIN {X 0.3271,Y -51.2583,Z 68,A -95.6732,B 24.8811,C -2.517,E1 25.0011,E2 539.3459} C_DIS
Startdeposition()
$VEL.CP = VEL_PRINT
LIN {X 1.4909,Y -50.3045,Z 68,A -93.6322,B 24.8783,C -2.5463,E1 25.007,E2 537.2357} C_DIS
LIN {X 4.7518,Y -50.1019,Z 68,A -90.0404,B 24.8783,C -2.5457,E1 25.017,E2 533.6471} C_DIS
LIN {X 7.1244,Y -49.8197,Z 68,A -87.1403,B 24.8779,C -2.5507,E1 25.0251,E2 530.7375} C_DIS
LIN {X 9.7513,Y -49.3734,Z 68,A -84.1791,B 24.8778,C -2.5518,E1 25.0332,E2 527.777} C_DIS
LIN {X 13.077,Y -48.5979,Z 68,A -79.8465,B 24.8766,C -2.5639,E1 25.045,E2 523.422} C_DIS
LIN {X 16.2764,Y -47.6223,Z 68,A -76.4835,B 24.877,C -2.56,E1 25.0539,E2 520.0745} C_DIS
LIN {X 18.7738,Y -46.6942,Z 68,A -73.3044,B 24.8763,C -2.5669,E1 25.0622,E2 516.8862} C_DIS
LIN {X 21.7147,Y -45.4009,Z 68,A -70.1036,B 24.8766,C -2.5637,E1 25.0703,E2 513.7009} C_DIS
LIN {X 23.5859,Y -44.4578,Z 68,A -67.405,B 24.8756,C -2.5736,E1 25.077,E2 510.9863} C_DIS
LIN {X 26.0107,Y -43.0839,Z 68,A -64.1192,B 24.8749,C -2.5815,E1 25.085,E2 507.6919} C_DIS
LIN {X 29.1966,Y -40.9918,Z 68,A -59.4692,B 24.8735,C -2.5961,E1 25.0957,E2 503.023} C_DIS
LIN {X 31.5221,Y -39.2322,Z 68,A -56.8415,B 24.8741,C -2.5895,E1 25.1014,E2 500.4208} C_DIS
LIN {X 33.4775,Y -37.577,Z 68,A -53.5824,B 24.8728,C -2.6028,E1 25.1083,E2 497.1429} C_DIS
LIN {X 35.3044,Y -35.866,Z 68,A -51.064,B 24.8728,C -2.6028,E1 25.1134,E2 494.6348} C_DIS
LIN {X 37.1049,Y -33.9999,Z 68,A -48.4775,B 24.8728,C -2.6028,E1 25.1184,E2 492.0598} C_DIS
LIN {X 38.2291,Y -32.7309,Z 68,A -46.276,B 24.8718,C -2.613,E1 25.1224,E2 489.8439} C_DIS
LIN {X 39.2453,Y -31.5059,Z 68,A -43.7359,B 24.8699,C -2.6325,E1 25.1269,E2 487.2695} C_DIS
LIN {X 41.8575,Y -27.9427,Z 68,A -39.0342,B 24.8692,C -2.6393,E1 25.1345,E2 482.5746} C_DIS
LIN {X 43.4374,Y -25.4163,Z 68,A -35.6907,B 24.8683,C -2.6479,E1 25.1393,E2 479.228} C_DIS
LIN {X 44.6798,Y -23.1638,Z 68,A -32.8906,B 24.8678,C -2.6537,E1 25.143,E2 476.4289} C_DIS
LIN {X 46.1748,Y -20.0164,Z 68,A -29.0431,B 24.8668,C -2.6629,E1 25.1474,E2 472.5803} C_DIS
LIN {X 47.1053,Y -17.7162,Z 68,A -25.939,B 24.8654,C -2.6772,E1 25.1506,E2 469.4597} C_DIS
LIN {X 47.9528,Y -15.2756,Z 68,A -23.2965,B 24.8651,C -2.68,E1 25.1529,E2 466.8255} C_DIS
LIN {X 48.6853,Y -12.7499,Z 68,A -19.5583,B 24.8626,C -2.7048,E1 25.1556,E2 463.0502} C_DIS
LIN {X 49.3802,Y -9.7161,Z 68,A -16.7835,B 24.8631,C -2.6998,E1 25.1572,E2 460.3033} C_DIS
LIN {X 49.8278,Y -7.0676,Z 68,A -13.7746,B 24.8622,C -2.7085,E1 25.1585,E2 457.2917} C_DIS
LIN {X 50.2646,Y -2.5106,Z 68,A -8.8087,B 24.8611,C -2.7198,E1 25.1596,E2 452.3285} C_DIS
LIN {X 50.3192,Y 0.8598,Z 68,A -4.7277,B 24.8593,C -2.7369,E1 25.1597,E2 448.2314} C_DIS
LIN {X 50.195,Y 3.6455,Z 68,A -1.5712,B 24.8583,C -2.7464,E1 25.1592,E2 445.071} C_DIS
LIN {X 49.922,Y 6.3693,Z 68,A 1.8468,B 24.8567,C -2.7623,E1 25.1581,E2 441.6356} C_DIS
LIN {X 49.3141,Y 10.0444,Z 68,A 5.7326,B 24.8561,C -2.768,E1 25.1561,E2 437.7592} C_DIS
LIN {X 48.7372,Y 12.5478,Z 68,A 8.6464,B 24.8552,C -2.7765,E1 25.1542,E2 434.842} C_DIS
LIN {X 48.0125,Y 15.0865,Z 68,A 11.5067,B 24.8546,C -2.7824,E1 25.1519,E2 431.9841} C_DIS
LIN {X 47.1929,Y 17.4831,Z 68,A 14.4389,B 24.8536,C -2.7918,E1 25.1491,E2 429.0462} C_DIS
LIN {X 45.8031,Y 20.8537,Z 68,A 18.57,B 24.8524,C -2.803,E1 25.1446,E2 424.9111} C_DIS
LIN {X 44.5267,Y 23.4549,Z 68,A 21.9921,B 24.8512,C -2.8145,E1 25.1403,E2 421.4801} C_DIS
LIN {X 43.1817,Y 25.8492,Z 68,A 24.9018,B 24.8508,C -2.8183,E1 25.1362,E2 418.5764} C_DIS
LIN {X 41.8082,Y 28.016,Z 68,A 28.4857,B 24.8486,C -2.8389,E1 25.1306,E2 414.9615} C_DIS
LIN {X 39.6886,Y 30.9461,Z 68,A 31.972,B 24.8489,C -2.8362,E1 25.1248,E2 411.4983} C_DIS
LIN {X 37.4905,Y 33.5742,Z 68,A 35.4089,B 24.8489,C -2.8359,E1 25.1186,E2 408.0777} C_DIS
LIN {X 34.823,Y 36.3338,Z 68,A 40.1966,B 24.8471,C -2.8532,E1 25.1092,E2 403.2695} C_DIS
LIN {X 32.3185,Y 38.5787,Z 68,A 43.6492,B 24.8471,C -2.8532,E1 25.102,E2 399.8303} C_DIS
LIN {X 29.3029,Y 40.9159,Z 68,A 48.3708,B 24.8455,C -2.868,E1 25.0914,E2 395.0908} C_DIS
LIN {X 26.9517,Y 42.5023,Z 68,A 51.8772,B 24.8443,C -2.8783,E1 25.0832,E2 391.5716} C_DIS
LIN {X 23.9712,Y 44.2509,Z 68,A 55.4881,B 24.8444,C -2.8776,E1 25.0745,E2 387.973} C_DIS
LIN {X 21.6521,Y 45.4309,Z 68,A 58.3647,B 24.8442,C -2.8796,E1 25.0673,E2 385.0993} C_DIS
LIN {X 18.96,Y 46.6184,Z 68,A 61.6891,B 24.8439,C -2.8827,E1 25.0587,E2 381.7755} C_DIS
LIN {X 16.7605,Y 47.4537,Z 68,A 64.3043,B 24.8437,C -2.8839,E1 25.0519,E2 379.1628} C_DIS
LIN {X 15.2216,Y 47.9702,Z 68,A 66.96,B 24.842,C -2.9,E1 25.0447,E2 376.4738} C_DIS
LIN {X 10.1083,Y 49.3009,Z 68,A 72.3349,B 24.8429,C -2.8917,E1 25.0302,E2 371.1263} C_DIS
LIN {X 7.5784,Y 49.7528,Z 68,A 75.2221,B 24.8429,C -2.892,E1 25.0222,E2 368.2415} C_DIS
LIN {X 4.5067,Y 50.1245,Z 68,A 78.8496,B 24.8426,C -2.8943,E1 25.0122,E2 364.6108} C_DIS
LIN {X 2.195,Y 50.2787,Z 68,A 81.3005,B 24.843,C -2.891,E1 25.0054,E2 362.1686} C_DIS
LIN {X -0.2121,Y 50.3262,Z 68,A 84.0153,B 24.843,C -2.8901,E1 24.9978,E2 359.4563} C_DIS
LIN {X -2.389,Y 50.2703,Z 68,A 87.1085,B 24.842,C -2.8997,E1 24.9891,E2 356.3395} C_DIS
LIN {X -5.2325,Y 50.0538,Z 68,A 90.392,B 24.8421,C -2.8987,E1 24.98,E2 353.0566} C_DIS
LIN {X -8.6003,Y 49.587,Z 68,A 93.6538,B 24.8435,C -2.8859,E1 24.971,E2 349.8223} C_DIS
LIN {X -10.8579,Y 49.1415,Z 68,A 96.3704,B 24.8435,C -2.8853,E1 24.9636,E2 347.104} C_DIS
LIN {X -13.4091,Y 48.5081,Z 68,A 99.3596,B 24.8439,C -2.8823,E1 24.9555,E2 344.1175} C_DIS
LIN {X -16.3015,Y 47.6138,Z 68,A 103.0194,B 24.8439,C -2.8818,E1 24.9458,E2 340.4523} C_DIS
LIN {X -18.9199,Y 46.6348,Z 68,A 106.4405,B 24.844,C -2.8814,E1 24.9369,E2 337.0247} C_DIS
LIN {X -21.7905,Y 45.3645,Z 68,A 109.7001,B 24.8451,C -2.871,E1 24.9287,E2 333.7817} C_DIS
LIN {X -23.8303,Y 44.3273,Z 68,A 112.0879,B 24.846,C -2.8634,E1 24.9228,E2 331.4056} C_DIS
LIN {X -25.7887,Y 43.2175,Z 68,A 114.6959,B 24.8464,C -2.8596,E1 24.9165,E2 328.7987} C_DIS
LIN {X -27.8291,Y 41.9324,Z 68,A 117.8813,B 24.8462,C -2.8612,E1 24.9091,E2 325.5992} C_DIS
LIN {X -30.4221,Y 40.091,Z 68,A 121.2562,B 24.8474,C -2.8501,E1 24.9015,E2 322.2387} C_DIS
LIN {X -32.5556,Y 38.3784,Z 68,A 124.3298,B 24.8482,C -2.8428,E1 24.8949,E2 319.171} C_DIS
LIN {X -34.5521,Y 36.5913,Z 68,A 127.4158,B 24.8489,C -2.8364,E1 24.8886,E2 316.0877} C_DIS
LIN {X -36.3665,Y 34.7887,Z 68,A 130.1551,B 24.8499,C -2.8269,E1 24.8832,E2 313.3594} C_DIS
LIN {X -37.842,Y 33.177,Z 68,A 132.9331,B 24.8501,C -2.8251,E1 24.878,E2 310.5735} C_DIS
LIN {X -39.147,Y 31.6272,Z 68,A 135.1254,B 24.8509,C -2.8175,E1 24.8742,E2 308.3891} C_DIS
LIN {X -40.7768,Y 29.4974,Z 68,A 138.2755,B 24.8516,C -2.8108,E1 24.8689,E2 305.2398} C_DIS
LIN {X -42.3455,Y 27.196,Z 68,A 141.3409,B 24.8527,C -2.8006,E1 24.8642,E2 302.1833} C_DIS
LIN {X -43.8946,Y 24.6177,Z 68,A 144.2226,B 24.8545,C -2.7832,E1 24.8602,E2 299.3283} C_DIS
LIN {X -45.187,Y 22.1573,Z 68,A 147.9901,B 24.8545,C -2.7827,E1 24.8553,E2 295.542} C_DIS
LIN {X -46.304,Y 19.7164,Z 68,A 151.6239,B 24.8546,C -2.782,E1 24.8512,E2 291.8899} C_DIS
LIN {X -47.5774,Y 16.4082,Z 68,A 155.1145,B 24.8567,C -2.762,E1 24.8479,E2 288.4274} C_DIS
LIN {X -48.5359,Y 13.3064,Z 68,A 159.3115,B 24.8572,C -2.7577,E1 24.8446,E2 284.2162} C_DIS
LIN {X -49.3165,Y 10.0325,Z 68,A 163.3177,B 24.8581,C -2.7483,E1 24.8423,E2 280.2091} C_DIS
LIN {X -50.0343,Y 5.4137,Z 68,A 168.1076,B 24.8606,C -2.724,E1 24.8405,E2 275.4487} C_DIS
LIN {X -50.2413,Y 2.9324,Z 68,A 171.3165,B 24.861,C -2.7204,E1 24.8399,E2 272.2291} C_DIS
LIN {X -50.3278,Y -0.1932,Z 68,A 174.6631,B 24.8625,C -2.7061,E1 24.8399,E2 268.8965} C_DIS
LIN {X -50.245,Y -2.8656,Z 68,A 177.6457,B 24.8635,C -2.6958,E1 24.8402,E2 265.9207} C_DIS
LIN {X -49.8943,Y -6.5831,Z 68,A -178.1522,B 24.8649,C -2.6819,E1 24.8414,E2 261.7267} C_DIS
LIN {X -49.4527,Y -9.3391,Z 68,A -174.9121,B 24.8658,C -2.673,E1 24.843,E2 258.4885} C_DIS
LIN {X -48.9749,Y -11.5886,Z 68,A -172.3717,B 24.8667,C -2.664,E1 24.8445,E2 255.9548} C_DIS
LIN {X -48.0266,Y -15.0407,Z 68,A -168.1595,B 24.8677,C -2.6539,E1 24.8478,E2 251.7424} C_DIS
LIN {X -47.1935,Y -17.4814,Z 68,A -165.1725,B 24.8685,C -2.6461,E1 24.8506,E2 248.757} C_DIS
LIN {X -45.8359,Y -20.7808,Z 68,A -160.9564,B 24.8694,C -2.637,E1 24.8552,E2 244.5394} C_DIS
LIN {X -44.6302,Y -23.2584,Z 68,A -158.0124,B 24.8706,C -2.6257,E1 24.8589,E2 241.6067} C_DIS
LIN {X -43.4655,Y -25.3691,Z 68,A -155.2685,B 24.8713,C -2.6184,E1 24.8627,E2 238.8658} C_DIS
LIN {X -41.8481,Y -27.9569,Z 68,A -151.8665,B 24.8722,C -2.6086,E1 24.8678,E2 235.4701} C_DIS
LIN {X -40.2365,Y -30.2289,Z 68,A -148.795,B 24.8731,C -2.5994,E1 24.8728,E2 232.4055} C_DIS
LIN {X -38.9791,Y -31.8344,Z 68,A -146.1844,B 24.8732,C -2.5984,E1 24.8774,E2 229.7851} C_DIS
LIN {X -36.8074,Y -34.3223,Z 68,A -142.7388,B 24.8745,C -2.5853,E1 24.8838,E2 226.3553} C_DIS
LIN {X -35.0556,Y -36.1095,Z 68,A -139.6907,B 24.8748,C -2.5825,E1 24.8898,E2 223.3011} C_DIS
LIN {X -33.288,Y -37.7456,Z 68,A -136.2742,B 24.8743,C -2.5877,E1 24.897,E2 219.8585} C_DIS
LIN {X -31.2328,Y -39.4623,Z 68,A -133.6509,B 24.8755,C -2.5755,E1 24.9026,E2 217.2545} C_DIS
LIN {X -28.6046,Y -41.4072,Z 68,A -129.9809,B 24.8761,C -2.5685,E1 24.9109,E2 213.5885} C_DIS
LIN {X -26.5573,Y -42.7491,Z 68,A -127.1615,B 24.8765,C -2.5648,E1 24.9176,E2 210.7687} C_DIS
LIN {X -24.1745,Y -44.1406,Z 68,A -123.9797,B 24.8768,C -2.5612,E1 24.9253,E2 207.5862} C_DIS
LIN {X -21.5468,Y -45.4812,Z 68,A -119.9527,B 24.8762,C -2.5683,E1 24.9355,E2 203.532} C_DIS
LIN {X -18.2919,Y -46.8848,Z 68,A -115.896,B 24.8765,C -2.5648,E1 24.946,E2 199.4747} C_DIS
LIN {X -13.1665,Y -48.5737,Z 68,A -110.4074,B 24.878,C -2.5493,E1 24.9606,E2 194.0135} C_DIS
LIN {X -10.6643,Y -49.1837,Z 68,A -107.516,B 24.8782,C -2.5472,E1 24.9684,E2 191.1234} C_DIS
LIN {X -7.5343,Y -49.7596,Z 68,A -103.6681,B 24.8779,C -2.55,E1 24.9791,E2 187.2652} C_DIS
LIN {X -4.8171,Y -50.0958,Z 68,A -100.8774,B 24.8785,C -2.5439,E1 24.9868,E2 184.4871} C_DIS
LIN {X -2.2453,Y -50.2765,Z 68,A -97.8304,B 24.8783,C -2.546,E1 24.9953,E2 181.4342} C_DIS
LIN {X 0.3217,Y -50.3112,Z 68,A -95.6763,B 24.8795,C -2.5333,E1 25.0012,E2 179.3104} C_DIS
Enddeposition()
LIN {X 0.3217,Y -50.3112,Z 68,A -95.6763,B 24.8795,C -2.5333,E1 25.0012,E2 179.3104} C_DIS
Startdeposition()
$VEL.CP = VEL_PRINT
LIN {X 0.0111,Y -49.3836,Z 68,A -96.8477,B 24.8793,C -2.5354,E1 24.998,E2 180.4768} C_DIS
LIN {X -2.7783,Y -49.3046,Z 68,A -99.8665,B 24.879,C -2.5388,E1 24.9896,E2 183.4881} C_DIS
LIN {X -5.2397,Y -49.1041,Z 68,A -102.6141,B 24.8788,C -2.5409,E1 24.9819,E2 186.232} C_DIS
LIN {X -6.9933,Y -48.8851,Z 68,A -104.9251,B 24.8792,C -2.537,E1 24.9755,E2 188.5541} C_DIS
LIN {X -9.7501,Y -48.411,Z 68,A -107.9752,B 24.8788,C -2.5413,E1 24.9672,E2 191.5972} C_DIS
LIN {X -12.0798,Y -47.8831,Z 68,A -110.7897,B 24.8787,C -2.542,E1 24.9595,E2 194.4138} C_DIS
LIN {X -14.6536,Y -47.1586,Z 68,A -114.3603,B 24.8792,C -2.5366,E1 24.9499,E2 198.0032} C_DIS
LIN {X -17.5766,Y -46.149,Z 68,A -117.6039,B 24.8784,C -2.5451,E1 24.9414,E2 201.233} C_DIS
LIN {X -20.2981,Y -45.0183,Z 68,A -121.0051,B 24.878,C -2.549,E1 24.9327,E2 204.633} C_DIS
LIN {X -22.5576,Y -43.9297,Z 68,A -124.0093,B 24.8778,C -2.551,E1 24.9252,E2 207.6403} C_DIS
LIN {X -25.0326,Y -42.5681,Z 68,A -127.3127,B 24.8774,C -2.555,E1 24.9172,E2 210.9438} C_DIS
LIN {X -27.4482,Y -41.0529,Z 68,A -130.6759,B 24.877,C -2.5592,E1 24.9093,E2 214.3079} C_DIS
LIN {X -29.6777,Y -39.4702,Z 68,A -133.7953,B 24.8765,C -2.5653,E1 24.9022,E2 217.4237} C_DIS
LIN {X -31.8809,Y -37.7134,Z 68,A -137.0541,B 24.8759,C -2.5714,E1 24.8952,E2 220.6802} C_DIS
LIN {X -33.7835,Y -36.0186,Z 68,A -140.0258,B 24.8753,C -2.577,E1 24.8891,E2 223.6506} C_DIS
LIN {X -35.6156,Y -34.2081,Z 68,A -142.6897,B 24.8743,C -2.588,E1 24.8839,E2 226.2997} C_DIS
LIN {X -37.0828,Y -32.6122,Z 68,A -145.5845,B 24.8743,C -2.588,E1 24.8784,E2 229.2074} C_DIS
LIN {X -38.7693,Y -30.5876,Z 68,A -148.6369,B 24.8736,C -2.5951,E1 24.8731,E2 232.2571} C_DIS
LIN {X -40.0889,Y -28.8371,Z 68,A -151.2831,B 24.8731,C -2.5997,E1 24.8687,E2 234.9049} C_DIS
LIN {X -41.5828,Y -26.637,Z 68,A -154.1384,B 24.872,C -2.6107,E1 24.8643,E2 237.7483} C_DIS
LIN {X -42.6405,Y -24.9101,Z 68,A -156.7487,B 24.8718,C -2.6131,E1 24.8606,E2 240.3663} C_DIS
LIN {X -43.8136,Y -22.7836,Z 68,A -159.5875,B 24.8711,C -2.6203,E1 24.8569,E2 243.2029} C_DIS
LIN {X -44.7994,Y -20.7768,Z 68,A -162.2464,B 24.8705,C -2.6266,E1 24.8537,E2 245.8613} C_DIS
LIN {X -45.8939,Y -18.2332,Z 68,A -165.4165,B 24.8695,C -2.6362,E1 24.8503,E2 249.026} C_DIS
LIN {X -46.7686,Y -15.8545,Z 68,A -168.2942,B 24.8686,C -2.6456,E1 24.8477,E2 251.8976} C_DIS
LIN {X -47.7967,Y -12.4158,Z 68,A -172.8219,B 24.8678,C -2.653,E1 24.8442,E2 256.4338} C_DIS
LIN {X -48.3654,Y -9.9723,Z 68,A -176.3178,B 24.8678,C -2.6541,E1 24.8422,E2 259.9479} C_DIS
LIN {X -49.0258,Y -5.9299,Z 68,A 179.5619,B 24.8654,C -2.6771,E1 24.8406,E2 264.0376} C_DIS
LIN {X -49.2989,Y -2.8814,Z 68,A 176.4069,B 24.8638,C -2.6935,E1 24.84,E2 267.1724} C_DIS
LIN {X -49.3826,Y -0.3468,Z 68,A 173.37,B 24.8629,C -2.7014,E1 24.8398,E2 270.2086} C_DIS
LIN {X -49.2258,Y 3.9342,Z 68,A 168.5677,B 24.8611,C -2.7194,E1 24.8404,E2 274.9969} C_DIS
LIN {X -48.8094,Y 7.5037,Z 68,A 163.227,B 24.8614,C -2.7169,E1 24.8424,E2 280.3754} C_DIS
LIN {X -48.2259,Y 10.6268,Z 68,A 159.9383,B 24.8597,C -2.7336,E1 24.8443,E2 283.6435} C_DIS
LIN {X -47.2389,Y 14.3947,Z 68,A 155.6805,B 24.8579,C -2.751,E1 24.8475,E2 287.8843} C_DIS
LIN {X -46.4339,Y 16.8097,Z 68,A 152.1292,B 24.8578,C -2.752,E1 24.8508,E2 291.4535} C_DIS
LIN {X -45.1234,Y 20.0648,Z 68,A 148.8514,B 24.8554,C -2.7747,E1 24.8543,E2 294.695} C_DIS
LIN {X -44.0851,Y 22.2537,Z 68,A 145.9958,B 24.8546,C -2.7823,E1 24.8578,E2 297.548} C_DIS
LIN {X -43.0615,Y 24.1739,Z 68,A 143.3481,B 24.854,C -2.7878,E1 24.8614,E2 300.1963} C_DIS
LIN {X -41.4118,Y 26.9035,Z 68,A 139.5721,B 24.853,C -2.7971,E1 24.8669,E2 303.9697} C_DIS
LIN {X -39.923,Y 29.0659,Z 68,A 136.5369,B 24.8522,C -2.8054,E1 24.8718,E2 306.9998} C_DIS
LIN {X -38.3423,Y 31.1211,Z 68,A 133.8035,B 24.8509,C -2.817,E1 24.8765,E2 309.7183} C_DIS
LIN {X -36.8671,Y 32.8555,Z 68,A 130.5456,B 24.8511,C -2.815,E1 24.8825,E2 312.9958} C_DIS
LIN {X -34.6615,Y 35.1744,Z 68,A 127.1605,B 24.8497,C -2.8284,E1 24.8891,E2 316.3631} C_DIS
LIN {X -32.833,Y 36.8873,Z 68,A 124.2164,B 24.8491,C -2.8345,E1 24.8952,E2 319.3047} C_DIS
LIN {X -30.8856,Y 38.5333,Z 68,A 121.4405,B 24.8481,C -2.8435,E1 24.9011,E2 322.0697} C_DIS
LIN {X -29.1384,Y 39.87,Z 68,A 118.6257,B 24.8479,C -2.8449,E1 24.9074,E2 324.8912} C_DIS
LIN {X -26.8198,Y 41.4655,Z 68,A 115.5543,B 24.847,C -2.854,E1 24.9145,E2 327.9512} C_DIS
LIN {X -24.7662,Y 42.7239,Z 68,A 112.7379,B 24.8465,C -2.8586,E1 24.9213,E2 330.765} C_DIS
LIN {X -22.5921,Y 43.9121,Z 68,A 109.7461,B 24.8461,C -2.8616,E1 24.9286,E2 333.7581} C_DIS
LIN {X -20.2805,Y 45.0262,Z 68,A 106.6859,B 24.8458,C -2.8648,E1 24.9364,E2 336.8181} C_DIS
LIN {X -18.1486,Y 45.9271,Z 68,A 104.4632,B 24.8446,C -2.8756,E1 24.9421,E2 339.0204} C_DIS
LIN {X -16.1508,Y 46.6672,Z 68,A 101.61,B 24.8449,C -2.8728,E1 24.9496,E2 341.8859} C_DIS
LIN {X -13.746,Y 47.4319,Z 68,A 98.5043,B 24.8449,C -2.8733,E1 24.9579,E2 344.9957} C_DIS
LIN {X -11.0685,Y 48.1264,Z 68,A 95.4883,B 24.8442,C -2.8793,E1 24.9661,E2 348.0015} C_DIS
LIN {X -8.6254,Y 48.6238,Z 68,A 92.416,B 24.8442,C -2.8787,E1 24.9745,E2 351.0786} C_DIS
LIN {X -6.7246,Y 48.9233,Z 68,A 90.2983,B 24.8439,C -2.882,E1 24.9803,E2 353.1902} C_DIS
LIN {X -4.6985,Y 49.159,Z 68,A 87.7873,B 24.8441,C -2.8809,E1 24.9873,E2 355.7053} C_DIS
LIN {X -2.1101,Y 49.3377,Z 68,A 84.8385,B 24.8438,C -2.883,E1 24.9955,E2 358.6499} C_DIS
LIN {X 0.2943,Y 49.3819,Z 68,A 82.2174,B 24.8435,C -2.8863,E1 25.0028,E2 361.2631} C_DIS
LIN {X 2.7824,Y 49.3044,Z 68,A 79.2051,B 24.8437,C -2.8845,E1 25.0112,E2 364.279} C_DIS
LIN {X 5.374,Y 49.0901,Z 68,A 76.0992,B 24.8439,C -2.8827,E1 25.0199,E2 367.3872} C_DIS
LIN {X 7.7951,Y 48.7643,Z 68,A 73.2401,B 24.8439,C -2.8815,E1 25.0278,E2 370.2465} C_DIS
LIN {X 10.1182,Y 48.3355,Z 68,A 70.375,B 24.8444,C -2.8782,E1 25.0356,E2 373.116} C_DIS
LIN {X 13.6404,Y 47.4619,Z 68,A 66.3448,B 24.8443,C -2.8787,E1 25.0465,E2 377.1387} C_DIS
LIN {X 15.8535,Y 46.7689,Z 68,A 63.3609,B 24.8451,C -2.8715,E1 25.0544,E2 380.134} C_DIS
LIN {X 18.8392,Y 45.6487,Z 68,A 60.0377,B 24.8448,C -2.8745,E1 25.063,E2 383.4426} C_DIS
LIN {X 21.2002,Y 44.601,Z 68,A 56.9968,B 24.8452,C -2.8703,E1 25.0707,E2 386.4858} C_DIS
LIN {X 23.5967,Y 43.3804,Z 68,A 53.8323,B 24.8457,C -2.8655,E1 25.0786,E2 389.6528} C_DIS
LIN {X 25.6148,Y 42.2201,Z 68,A 51.4474,B 24.8455,C -2.8673,E1 25.0843,E2 392.026} C_DIS
LIN {X 27.3322,Y 41.1296,Z 68,A 48.783,B 24.8465,C -2.8582,E1 25.0905,E2 394.7034} C_DIS
LIN {X 29.8864,Y 39.3131,Z 68,A 45.2509,B 24.847,C -2.8539,E1 25.0985,E2 398.2331} C_DIS
LIN {X 31.9572,Y 37.6485,Z 68,A 42.1328,B 24.8477,C -2.8476,E1 25.1052,E2 401.3543} C_DIS
LIN {X 33.8983,Y 35.9106,Z 68,A 39.587,B 24.8473,C -2.8505,E1 25.1104,E2 403.8829} C_DIS
LIN {X 35.4997,Y 34.3284,Z 68,A 36.5543,B 24.8488,C -2.8371,E1 25.1164,E2 406.9344} C_DIS
LIN {X 37.3034,Y 32.3595,Z 68,A 33.4168,B 24.8496,C -2.8295,E1 25.1223,E2 410.0759} C_DIS
LIN {X 39.0173,Y 30.271,Z 68,A 30.7479,B 24.8494,C -2.8311,E1 25.1269,E2 412.7286} C_DIS
LIN {X 40.3562,Y 28.4624,Z 68,A 27.7915,B 24.8508,C -2.8182,E1 25.1318,E2 415.7014} C_DIS
LIN {X 41.7468,Y 26.3804,Z 68,A 24.8035,B 24.8518,C -2.8092,E1 25.1364,E2 418.6956} C_DIS
LIN {X 43.081,Y 24.1391,Z 68,A 21.6754,B 24.8528,C -2.7993,E1 25.1407,E2 421.831} C_DIS
LIN {X 44.3504,Y 21.7193,Z 68,A 18.8744,B 24.853,C -2.7979,E1 25.1442,E2 424.6205} C_DIS
LIN {X 45.4607,Y 19.286,Z 68,A 15.1754,B 24.8551,C -2.7776,E1 25.1484,E2 428.3473} C_DIS
LIN {X 47.005,Y 15.139,Z 68,A 10.4781,B 24.8557,C -2.7713,E1 25.1528,E2 433.0331} C_DIS
LIN {X 47.7945,Y 12.4242,Z 68,A 7.2138,B 24.8567,C -2.7618,E1 25.1552,E2 436.3011} C_DIS
LIN {X 48.4269,Y 9.673,Z 68,A 3.968,B 24.8577,C -2.7525,E1 25.1571,E2 439.5502} C_DIS
LIN {X 48.845,Y 7.2732,Z 68,A 1.1383,B 24.8586,C -2.7437,E1 25.1584,E2 442.3839} C_DIS
LIN {X 49.1728,Y 4.5495,Z 68,A -1.9806,B 24.8595,C -2.7351,E1 25.1593,E2 445.5047} C_DIS
LIN {X 49.3517,Y 1.7711,Z 68,A -5.2319,B 24.8606,C -2.7246,E1 25.1597,E2 448.7616} C_DIS
LIN {X 49.3844,Y -0.1469,Z 68,A -7.6442,B 24.8617,C -2.7138,E1 25.1597,E2 451.185} C_DIS
LIN {X 49.3087,Y -2.7032,Z 68,A -10.5701,B 24.8626,C -2.7053,E1 25.1594,E2 454.1136} C_DIS
LIN {X 49.0521,Y -5.7051,Z 68,A -13.7801,B 24.8631,C -2.7,E1 25.1585,E2 457.3172} C_DIS
LIN {X 48.6868,Y -8.2625,Z 68,A -16.725,B 24.8639,C -2.6916,E1 25.1572,E2 460.2646} C_DIS
LIN {X 48.1983,Y -10.7534,Z 68,A -19.3915,B 24.8643,C -2.688,E1 25.1557,E2 462.9242} C_DIS
LIN {X 47.6862,Y -12.8332,Z 68,A -22.0928,B 24.8655,C -2.6759,E1 25.1538,E2 465.6383} C_DIS
LIN {X 47.0654,Y -14.9525,Z 68,A -24.5467,B 24.8661,C -2.6702,E1 25.1518,E2 468.0918} C_DIS
LIN {X 46.4696,Y -16.7119,Z 68,A -27.5627,B 24.8685,C -2.6466,E1 25.1489,E2 471.1467} C_DIS
LIN {X 45.0514,Y -20.2246,Z 68,A -31.0779,B 24.868,C -2.6509,E1 25.1451,E2 474.6325} C_DIS
LIN {X 44.1067,Y -22.211,Z 68,A -33.6722,B 24.8689,C -2.6426,E1 25.1419,E2 477.2326} C_DIS
LIN {X 43.186,Y -23.951,Z 68,A -36.1097,B 24.8698,C -2.633,E1 25.1387,E2 479.68} C_DIS
LIN {X 41.8073,Y -26.2831,Z 68,A -38.8183,B 24.8698,C -2.6327,E1 25.1348,E2 482.3754} C_DIS
LIN {X 40.9232,Y -27.6398,Z 68,A -41.1195,B 24.8712,C -2.6193,E1 25.1312,E2 484.697} C_DIS
LIN {X 39.0768,Y -30.1938,Z 68,A -44.8551,B 24.8723,C -2.6081,E1 25.1249,E2 488.4413} C_DIS
LIN {X 37.2112,Y -32.4651,Z 68,A -47.9539,B 24.8726,C -2.6054,E1 25.1193,E2 491.5322} C_DIS
LIN {X 34.886,Y -34.9527,Z 68,A -51.5977,B 24.8729,C -2.6017,E1 25.1123,E2 495.169} C_DIS
LIN {X 32.7936,Y -36.9226,Z 68,A -55.9649,B 24.8756,C -2.5744,E1 25.1032,E2 499.5833} C_DIS
LIN {X 29.6626,Y -39.4813,Z 68,A -60.3428,B 24.876,C -2.5704,E1 25.0936,E2 503.9545} C_DIS
LIN {X 26.7493,Y -41.5107,Z 68,A -64.041,B 24.876,C -2.5702,E1 25.0851,E2 507.6406} C_DIS
LIN {X 24.7294,Y -42.745,Z 68,A -66.6889,B 24.8763,C -2.5671,E1 25.0787,E2 510.2877} C_DIS
LIN {X 22.6838,Y -43.8652,Z 68,A -69.446,B 24.8768,C -2.5616,E1 25.0719,E2 513.05} C_DIS
LIN {X 20.535,Y -44.9115,Z 68,A -71.9014,B 24.8767,C -2.5631,E1 25.0657,E2 515.4955} C_DIS
LIN {X 18.4138,Y -45.8218,Z 68,A -74.8749,B 24.8776,C -2.5539,E1 25.058,E2 518.4839} C_DIS
LIN {X 15.8733,Y -46.7622,Z 68,A -77.9037,B 24.8777,C -2.552,E1 25.0501,E2 521.511} C_DIS
LIN {X 12.1873,Y -47.8554,Z 68,A -82.5013,B 24.8784,C -2.5447,E1 25.0377,E2 526.1182} C_DIS
LIN {X 9.624,Y -48.4368,Z 68,A -85.5093,B 24.8786,C -2.5428,E1 25.0295,E2 529.127} C_DIS
LIN {X 7.1155,Y -48.8678,Z 68,A -88.5099,B 24.8789,C -2.5398,E1 25.0212,E2 532.1316} C_DIS
LIN {X 4.9958,Y -49.1297,Z 68,A -90.8543,B 24.8789,C -2.5407,E1 25.0147,E2 534.4723} C_DIS
LIN {X 2.5943,Y -49.3148,Z 68,A -93.5679,B 24.8789,C -2.5409,E1 25.0072,E2 537.1843} C_DIS
LIN {X 0.3057,Y -49.3786,Z 68,A -95.0855,B 24.877,C -2.5598,E1 25.0031,E2 538.6565} C_DIS
Enddeposition()
LIN {X 0.3057,Y -49.3786,Z 68,A -95.0855,B 24.877,C -2.5598,E1 25.0031,E2 538.6565} C_DIS
Startdeposition()
$VEL.CP = VEL_PRINT
LIN {X 1.7712,Y -48.4075,Z 68,A -93.3293,B 24.8753,C -2.5768,E1 25.0081,E2 536.8603} C_DIS
LIN {X 4.1492,Y -48.2619,Z 68,A -90.4892,B 24.8752,C -2.5785,E1 25.016,E2 534.0176} C_DIS
LIN {X 6.4476,Y -48.0085,Z 68,A -87.7391,B 24.875,C -2.5805,E1 25.0236,E2 531.265} C_DIS
LIN {X 8.8611,Y -47.6225,Z 68,A -84.8991,B 24.8749,C -2.5818,E1 25.0314,E2 528.425} C_DIS
LIN {X 11.181,Y -47.1318,Z 68,A -82.0777,B 24.8746,C -2.5846,E1 25.0391,E2 525.6006} C_DIS
LIN {X 13.4033,Y -46.5482,Z 68,A -79.3416,B 24.8743,C -2.5878,E1 25.0465,E2 522.8613} C_DIS
LIN {X 15.6872,Y -45.829,Z 68,A -76.5169,B 24.874,C -2.5911,E1 25.054,E2 520.0342} C_DIS
LIN {X 17.9814,Y -44.9788,Z 68,A -73.6722,B 24.8737,C -2.5941,E1 25.0614,E2 517.1887} C_DIS
LIN {X 20.1779,Y -44.0372,Z 68,A -70.8409,B 24.8732,C -2.5984,E1 25.0686,E2 514.3541} C_DIS
LIN {X 22.308,Y -42.9975,Z 68,A -68.0672,B 24.8729,C -2.6023,E1 25.0756,E2 511.5785} C_DIS
LIN {X 24.3845,Y -41.8547,Z 68,A -65.2526,B 24.8724,C -2.6074,E1 25.0824,E2 508.7602} C_DIS
LIN {X 26.4019,Y -40.6123,Z 68,A -62.4594,B 24.8719,C -2.6125,E1 25.089,E2 505.964} C_DIS
LIN {X 28.354,Y -39.2742,Z 68,A -59.7001,B 24.8714,C -2.6174,E1 25.0953,E2 503.2027} C_DIS
LIN {X 30.2678,Y -37.8192,Z 68,A -56.858,B 24.8708,C -2.6233,E1 25.1016,E2 500.3569} C_DIS
LIN {X 32.0667,Y -36.3061,Z 68,A -54.0942,B 24.8702,C -2.6292,E1 25.1074,E2 497.59} C_DIS
LIN {X 33.8025,Y -34.6958,Z 68,A -51.1529,B 24.8693,C -2.6385,E1 25.1134,E2 494.639} C_DIS
LIN {X 35.6401,Y -32.8044,Z 68,A -47.999,B 24.8685,C -2.6468,E1 25.1194,E2 491.4791} C_DIS
LIN {X 37.444,Y -30.7306,Z 68,A -44.9598,B 24.868,C -2.6509,E1 25.1249,E2 488.444} C_DIS
LIN {X 38.8904,Y -28.8781,Z 68,A -42.2216,B 24.8674,C -2.6575,E1 25.1295,E2 485.7034} C_DIS
LIN {X 40.1959,Y -27.0306,Z 68,A -39.5522,B 24.8667,C -2.6646,E1 25.1338,E2 483.0302} C_DIS
LIN {X 41.4336,Y -25.0919,Z 68,A -36.7447,B 24.8657,C -2.6739,E1 25.1379,E2 480.2149} C_DIS
LIN {X 42.7203,Y -22.8343,Z 68,A -33.7983,B 24.8651,C -2.6802,E1 25.1419,E2 477.269} C_DIS
LIN {X 43.7548,Y -20.7824,Z 68,A -31.0764,B 24.8643,C -2.6882,E1 25.1452,E2 474.5428} C_DIS
LIN {X 44.7467,Y -18.5513,Z 68,A -28.2307,B 24.8635,C -2.696,E1 25.1484,E2 471.6943} C_DIS
LIN {X 45.5747,Y -16.4112,Z 68,A -25.476,B 24.8626,C -2.705,E1 25.1511,E2 468.9336} C_DIS
LIN {X 46.3323,Y -14.1317,Z 68,A -22.6651,B 24.8618,C -2.7131,E1 25.1535,E2 466.1195} C_DIS
LIN {X 46.9731,Y -11.8288,Z 68,A -19.8819,B 24.861,C -2.721,E1 25.1554,E2 463.3337} C_DIS
LIN {X 47.5101,Y -9.4453,Z 68,A -17.0365,B 24.8601,C -2.7291,E1 25.1571,E2 460.4856} C_DIS
LIN {X 47.9044,Y -7.1801,Z 68,A -14.2876,B 24.8592,C -2.7382,E1 25.1583,E2 457.7312} C_DIS
LIN {X 48.1984,Y -4.8269,Z 68,A -11.5266,B 24.8584,C -2.7462,E1 25.1592,E2 454.9678} C_DIS
LIN {X 48.3816,Y -2.3759,Z 68,A -8.6618,B 24.8575,C -2.7545,E1 25.1597,E2 452.1004} C_DIS
LIN {X 48.4388,Y -0.347,Z 68,A -6.3849,B 24.857,C -2.7596,E1 25.1597,E2 449.825} C_DIS
LIN {X 48.407,Y 1.7861,Z 68,A -3.7736,B 24.856,C -2.7693,E1 25.1596,E2 447.2062} C_DIS
LIN {X 48.2614,Y 4.1547,Z 68,A -0.9628,B 24.855,C -2.7781,E1 25.159,E2 444.3913} C_DIS
LIN {X 48.0093,Y 6.4413,Z 68,A 1.7637,B 24.8541,C -2.7867,E1 25.1581,E2 441.6607} C_DIS
LIN {X 47.6206,Y 8.8714,Z 68,A 4.6059,B 24.8533,C -2.7942,E1 25.1567,E2 438.8173} C_DIS
LIN {X 47.129,Y 11.1931,Z 68,A 7.4181,B 24.8524,C -2.8028,E1 25.155,E2 436.0011} C_DIS
LIN {X 46.5439,Y 13.4183,Z 68,A 10.1459,B 24.8516,C -2.811,E1 25.153,E2 433.2694} C_DIS
LIN {X 45.8244,Y 15.7008,Z 68,A 12.9548,B 24.8507,C -2.8189,E1 25.1505,E2 430.4579} C_DIS
LIN {X 44.9803,Y 17.9776,Z 68,A 15.7624,B 24.85,C -2.8258,E1 25.1477,E2 427.6495} C_DIS
LIN {X 44.0541,Y 20.1406,Z 68,A 18.5485,B 24.8492,C -2.8336,E1 25.1445,E2 424.86} C_DIS
LIN {X 43.0326,Y 22.2391,Z 68,A 21.2807,B 24.8484,C -2.8406,E1 25.1411,E2 422.126} C_DIS
LIN {X 41.8508,Y 24.3914,Z 68,A 24.1843,B 24.8476,C -2.8482,E1 25.1371,E2 419.2193} C_DIS
LIN {X 40.6066,Y 26.4108,Z 68,A 26.9743,B 24.8469,C -2.8551,E1 25.1329,E2 416.4272} C_DIS
LIN {X 39.2653,Y 28.3665,Z 68,A 29.7406,B 24.8462,C -2.8612,E1 25.1285,E2 413.6599} C_DIS
LIN {X 37.8188,Y 30.2682,Z 68,A 32.5443,B 24.8455,C -2.8674,E1 25.1237,E2 410.8546} C_DIS
LIN {X 36.2867,Y 32.089,Z 68,A 35.3631,B 24.8448,C -2.8738,E1 25.1185,E2 408.0334} C_DIS
LIN {X 34.7,Y 33.7981,Z 68,A 38.1198,B 24.8442,C -2.8797,E1 25.1132,E2 405.2747} C_DIS
LIN {X 32.9955,Y 35.4641,Z 68,A 40.9274,B 24.8436,C -2.8852,E1 25.1075,E2 402.4657} C_DIS
LIN {X 31.1863,Y 37.0654,Z 68,A 43.7611,B 24.843,C -2.8902,E1 25.1015,E2 399.6313} C_DIS
LIN {X 29.3657,Y 38.5235,Z 68,A 46.5077,B 24.8425,C -2.8949,E1 25.0955,E2 396.8837} C_DIS
LIN {X 27.4058,Y 39.9418,Z 68,A 49.3502,B 24.8421,C -2.8992,E1 25.089,E2 394.0407} C_DIS
LIN {X 25.4053,Y 41.2431,Z 68,A 52.1838,B 24.8416,C -2.9037,E1 25.0823,E2 391.2057} C_DIS
LIN {X 23.4188,Y 42.4023,Z 68,A 54.9214,B 24.8411,C -2.9078,E1 25.0757,E2 388.4665} C_DIS
LIN {X 21.2496,Y 43.5302,Z 68,A 57.7815,B 24.8408,C -2.9108,E1 25.0685,E2 385.6071} C_DIS
LIN {X 19.0929,Y 44.5183,Z 68,A 60.558,B 24.8405,C -2.9133,E1 25.0615,E2 382.8313} C_DIS
LIN {X 16.9589,Y 45.3738,Z 68,A 63.302,B 24.8402,C -2.9163,E1 25.0543,E2 380.0861} C_DIS
LIN {X 14.6311,Y 46.1774,Z 68,A 66.2013,B 24.84,C -2.9184,E1 25.0466,E2 377.1874} C_DIS
LIN {X 12.4297,Y 46.8176,Z 68,A 68.9336,B 24.8397,C -2.9206,E1 25.0393,E2 374.4545} C_DIS
LIN {X 10.0629,Y 47.383,Z 68,A 71.7723,B 24.8397,C -2.9213,E1 25.0315,E2 371.6179} C_DIS
LIN {X 7.6983,Y 47.8243,Z 68,A 74.6067,B 24.8395,C -2.9221,E1 25.0237,E2 368.7846} C_DIS
LIN {X 5.3463,Y 48.144,Z 68,A 77.413,B 24.8395,C -2.9226,E1 25.016,E2 365.9793} C_DIS
LIN {X 3.105,Y 48.3397,Z 68,A 80.1476,B 24.8393,C -2.924,E1 25.0083,E2 363.2428} C_DIS
LIN {X 0.6685,Y 48.4349,Z 68,A 82.9823,B 24.8395,C -2.9228,E1 25.0004,E2 360.4114} C_DIS
LIN {X -1.7776,Y 48.4073,Z 68,A 85.855,B 24.8395,C -2.9217,E1 24.9924,E2 357.541} C_DIS
LIN {X -4.1466,Y 48.2621,Z 68,A 88.6512,B 24.8397,C -2.9204,E1 24.9847,E2 354.747} C_DIS
LIN {X -6.452,Y 48.008,Z 68,A 91.4603,B 24.8397,C -2.9198,E1 24.9769,E2 351.9372} C_DIS
LIN {X -8.867,Y 47.6215,Z 68,A 94.3108,B 24.8401,C -2.9171,E1 24.969,E2 349.0905} C_DIS
LIN {X -11.1889,Y 47.13,Z 68,A 97.1462,B 24.8403,C -2.915,E1 24.9613,E2 346.2562} C_DIS
LIN {X -13.414,Y 46.5451,Z 68,A 99.8987,B 24.8406,C -2.9127,E1 24.9539,E2 343.5049} C_DIS
LIN {X -15.6769,Y 45.8325,Z 68,A 102.677,B 24.841,C -2.909,E1 24.9465,E2 340.7303} C_DIS
LIN {X -17.7834,Y 45.0566,Z 68,A 105.3759,B 24.8413,C -2.9063,E1 24.9395,E2 338.0324} C_DIS
LIN {X -19.9316,Y 44.1483,Z 68,A 108.236,B 24.8416,C -2.9038,E1 24.9322,E2 335.1713} C_DIS
LIN {X -22.3113,Y 42.9957,Z 68,A 111.2352,B 24.8423,C -2.8969,E1 24.9247,E2 332.1806} C_DIS
LIN {X -24.3905,Y 41.8513,Z 68,A 114.0777,B 24.8428,C -2.8926,E1 24.9178,E2 329.34} C_DIS
LIN {X -26.4111,Y 40.6064,Z 68,A 116.8971,B 24.8433,C -2.8876,E1 24.9112,E2 326.5235} C_DIS
LIN {X -28.368,Y 39.2642,Z 68,A 119.7004,B 24.8439,C -2.8821,E1 24.9048,E2 323.7239} C_DIS
LIN {X -30.2712,Y 37.8164,Z 68,A 122.546,B 24.8445,C -2.8764,E1 24.8985,E2 320.8814} C_DIS
LIN {X -32.0858,Y 36.2895,Z 68,A 125.3677,B 24.8452,C -2.8705,E1 24.8926,E2 318.0629} C_DIS
LIN {X -33.7974,Y 34.7007,Z 68,A 128.1555,B 24.8458,C -2.8645,E1 24.8869,E2 315.2779} C_DIS
LIN {X -35.4546,Y 33.0057,Z 68,A 130.9749,B 24.8465,C -2.8579,E1 24.8815,E2 312.4619} C_DIS
LIN {X -37.067,Y 31.1843,Z 68,A 133.8569,B 24.8473,C -2.8508,E1 24.8763,E2 309.5839} C_DIS
LIN {X -38.527,Y 29.3611,Z 68,A 136.6371,B 24.8481,C -2.8439,E1 24.8715,E2 306.8071} C_DIS
LIN {X -39.9387,Y 27.4103,Z 68,A 139.4926,B 24.8489,C -2.8363,E1 24.8669,E2 303.9556} C_DIS
LIN {X -41.2321,Y 25.4231,Z 68,A 142.3376,B 24.8496,C -2.8291,E1 24.8627,E2 301.1133} C_DIS
LIN {X -42.4023,Y 23.4187,Z 68,A 145.1259,B 24.8504,C -2.822,E1 24.8588,E2 298.3276} C_DIS
LIN {X -43.5309,Y 21.2483,Z 68,A 148.0149,B 24.8513,C -2.8135,E1 24.8552,E2 295.4433} C_DIS
LIN {X -44.5196,Y 19.0901,Z 68,A 150.8272,B 24.8522,C -2.8053,E1 24.852,E2 292.6352} C_DIS
LIN {X -45.3816,Y 16.9381,Z 68,A 153.6011,B 24.853,C -2.7975,E1 24.8492,E2 289.8643} C_DIS
LIN {X -46.1754,Y 14.6375,Z 68,A 156.5007,B 24.8539,C -2.789,E1 24.8467,E2 286.9686} C_DIS
LIN {X -46.8145,Y 12.4413,Z 68,A 159.2499,B 24.8547,C -2.7813,E1 24.8447,E2 284.2219} C_DIS
LIN {X -47.389,Y 10.0352,Z 68,A 162.1471,B 24.8557,C -2.7718,E1 24.8429,E2 281.3304} C_DIS
LIN {X -47.8177,Y 7.7378,Z 68,A 164.9232,B 24.8566,C -2.7633,E1 24.8415,E2 278.5581} C_DIS
LIN {X -48.1298,Y 5.4672,Z 68,A 167.7023,B 24.8574,C -2.7557,E1 24.8406,E2 275.7805} C_DIS
LIN {X -48.3516,Y 2.92,Z 68,A 170.8531,B 24.8582,C -2.7479,E1 24.8399,E2 272.6295} C_DIS
LIN {X -48.4387,Y 0.3503,Z 68,A 173.6676,B 24.8595,C -2.7353,E1 24.8398,E2 269.8282} C_DIS
LIN {X -48.4071,Y -1.7837,Z 68,A 176.3208,B 24.8601,C -2.7291,E1 24.84,E2 267.1739} C_DIS
LIN {X -48.2615,Y -4.1538,Z 68,A 179.0978,B 24.8611,C -2.7199,E1 24.8405,E2 264.4021} C_DIS
LIN {X -48.008,Y -6.4518,Z 68,A -178.0331,B 24.8617,C -2.7133,E1 24.8415,E2 261.5317} C_DIS
LIN {X -47.6196,Y -8.8766,Z 68,A -175.1776,B 24.8627,C -2.7037,E1 24.8429,E2 258.6822} C_DIS
LIN {X -47.1309,Y -11.1848,Z 68,A -172.3396,B 24.8635,C -2.6959,E1 24.8446,E2 255.8461} C_DIS
LIN {X -46.5505,Y -13.3949,Z 68,A -169.5786,B 24.8642,C -2.6887,E1 24.8467,E2 253.0863} C_DIS
LIN {X -45.8287,Y -15.688,Z 68,A -166.7289,B 24.8651,C -2.6805,E1 24.8491,E2 250.24} C_DIS
LIN {X -44.9796,Y -17.9795,Z 68,A -163.8663,B 24.8659,C -2.6718,E1 24.852,E2 247.382} C_DIS
LIN {X -44.046,Y -20.1585,Z 68,A -161.0141,B 24.8667,C -2.6647,E1 24.8552,E2 244.5312} C_DIS
LIN {X -42.997,Y -22.3088,Z 68,A -158.1953,B 24.8674,C -2.6569,E1 24.8588,E2 241.716} C_DIS
LIN {X -41.8524,Y -24.3885,Z 68,A -155.3479,B 24.8681,C -2.6501,E1 24.8627,E2 238.8699} C_DIS
Enddeposition()
END
